// TIA Portal V20 program export: 2 tag tables, 2 data types, 3 data blocks, 5 code blocks (in call order from the OBs), 4 instance data blocks

VAR_GLOBAL   // PLC tag table "IO_Device_PCL_Centralilze_PLC_Functinal_Test_2"
   In_Test_Parameters AT %I100.0 : "IO_Device_Test_Parameters";
   Out_Functinal_Test AT %Q100.0 : "IO_Device_Functinal_Test";
END_VAR

VAR_GLOBAL   // PLC tag table "IO_PLC_Functinal_Test_2_PLC_Functinal_Test_4"
   In_Functional_Test AT %I300.0 : "IO_Device_Functinal_Test";
   Out_Test_Parameters AT %Q300.0 : "IO_Device_Test_Parameters";
END_VAR

TYPE "IO_Device_Functinal_Test"
   STRUCT
      Life_Trigger_PLC_Functional_Test_2 : Bool;
      Star_Test_PLC_Functional_Test_2 : Bool;
      Button_PLC_Functional_Test_2 : Bool;
      Electrical_Current_Test_Approved_PLC_Functional_Test_2 : Bool;
      Visual_Test_Approved_PLC_Functional_Test_2 : Bool;
      Electrical_Current_Read_PLC_Functional_Test_2 : UInt;
      Life_Trigger_PLC_Functional_Test_4 : Bool;
      Star_Test_PLC_Functional_Test_4 : Bool;
      Button_PLC_Functional_Test_4 : Bool;
      Electrical_Current_Test_Approved_PLC_Functional_Test_4 : Bool;
      Visual_Test_Approved_PLC_Functional_Test_4 : Bool;
      Electrical_Current_Read_PLC_Functional_Test_4 : UInt;
      Life_Trigger_PLC_Functional_Test_6 : Bool;
      Star_Test_PLC_Functional_Test_6 : Bool;
      Button_PLC_Functional_Test_6 : Bool;
      Electrical_Current_Test_Approved_PLC_Functional_Test_6 : Bool;
      Visual_Test_Approved_PLC_Functional_Test_6 : Bool;
      Electrical_Current_Read_PLC_Functional_Test_6 : UInt;
      Life_Trigger_PLC_Functional_Test_8 : Bool;
      Star_Test_PLC_Functional_Test_8 : Bool;
      Button_PLC_Functional_Test_8 : Bool;
      Electrical_Current_Test_Approved_PLC_Functional_Test_8 : Bool;
      Visual_Test_Approved_PLC_Functional_Test_8 : Bool;
      Electrical_Current_Read_PLC_Functional_Test_8 : UInt;
      Life_Trigger_PLC_Functional_Test_10 : Bool;
      Star_Test_PLC_Functional_Test_10 : Bool;
      Button_PLC_Functional_Test_10 : Bool;
      Electrical_Current_Test_Approved_PLC_Functional_Test_10 : Bool;
      Visual_Test_Approved_PLC_Functional_Test_10 : Bool;
      Electrical_Current_Read_PLC_Functional_Test_10 : UInt;
      Life_Trigger_PLC_Functional_Test_12 : Bool;
      Star_Test_PLC_Functional_Test_12 : Bool;
      Button_PLC_Functional_Test_12 : Bool;
      Electrical_Current_Test_Approved_PLC_Functional_Test_12 : Bool;
      Visual_Test_Approved_PLC_Functional_Test_12 : Bool;
      Electrical_Current_Read_PLC_Functional_Test_12 : UInt;
      Life_Trigger_PLC_Functional_Test_14 : Bool;
      Star_Test_PLC_Functional_Test_14 : Bool;
      Button_PLC_Functional_Test_14 : Bool;
      Electrical_Current_Test_Approved_PLC_Functional_Test_14 : Bool;
      Visual_Test_Approved_PLC_Functional_Test_14 : Bool;
      Electrical_Current_Read_PLC_Functional_Test_14 : UInt;
      Life_Trigger_PLC_Functional_Test_16 : Bool;
      Star_Test_PLC_Functional_Test_16 : Bool;
      Button_PLC_Functional_Test_16 : Bool;
      Electrical_Current_Test_Approved_PLC_Functional_Test_16 : Bool;
      Visual_Test_Approved_PLC_Functional_Test_16 : Bool;
      Electrical_Current_Read_PLC_Functional_Test_16 : UInt;
      Life_Trigger_PLC_Functional_Test_18 : Bool;
      Star_Test_PLC_Functional_Test_18 : Bool;
      Button_PLC_Functional_Test_18 : Bool;
      Electrical_Current_Test_Approved_PLC_Functional_Test_18 : Bool;
      Visual_Test_Approved_PLC_Functional_Test_18 : Bool;
      Electrical_Current_Read_PLC_Functional_Test_18 : UInt;
      Life_Trigger_PLC_Functional_Test_20 : Bool;
      Star_Test_PLC_Functional_Test_20 : Bool;
      Button_PLC_Functional_Test_20 : Bool;
      Electrical_Current_Test_Approved_PLC_Functional_Test_20 : Bool;
      Visual_Test_Approved_PLC_Functional_Test_20 : Bool;
      Electrical_Current_Read_PLC_Functional_Test_20 : UInt;
      Life_Trigger_PLC_Functional_Test_22 : Bool;
      Star_Test_PLC_Functional_Test_22 : Bool;
      Button_PLC_Functional_Test_22 : Bool;
      Electrical_Current_Test_Approved_PLC_Functional_Test_22 : Bool;
      Visual_Test_Approved_PLC_Functional_Test_22 : Bool;
      Electrical_Current_Read_PLC_Functional_Test_22 : UInt;
      Life_Trigger_PLC_Functional_Test_24 : Bool;
      Star_Test_PLC_Functional_Test_24 : Bool;
      Button_PLC_Functional_Test_24 : Bool;
      Electrical_Current_Test_Approved_PLC_Functional_Test_24 : Bool;
      Visual_Test_Approved_PLC_Functional_Test_24 : Bool;
      Electrical_Current_Read_PLC_Functional_Test_24 : UInt;
      Life_Trigger_PLC_Functional_Test_26 : Bool;
      Star_Test_PLC_Functional_Test_26 : Bool;
      Button_PLC_Functional_Test_26 : Bool;
      Electrical_Current_Test_Approved_PLC_Functional_Test_26 : Bool;
      Visual_Test_Approved_PLC_Functional_Test_26 : Bool;
      Electrical_Current_Read_PLC_Functional_Test_26 : UInt;
      Life_Trigger_PLC_Functional_Test_28 : Bool;
      Star_Test_PLC_Functional_Test_28 : Bool;
      Button_PLC_Functional_Test_28 : Bool;
      Electrical_Current_Test_Approved_PLC_Functional_Test_28 : Bool;
      Visual_Test_Approved_PLC_Functional_Test_28 : Bool;
      Electrical_Current_Read_PLC_Functional_Test_28 : UInt;
      Life_Trigger_PLC_Functional_Test_30 : Bool;
      Star_Test_PLC_Functional_Test_30 : Bool;
      Button_PLC_Functional_Test_30 : Bool;
      Electrical_Current_Test_Approved_PLC_Functional_Test_30 : Bool;
      Visual_Test_Approved_PLC_Functional_Test_30 : Bool;
      Electrical_Current_Read_PLC_Functional_Test_30 : UInt;
   END_STRUCT;
END_TYPE

TYPE "IO_Device_Test_Parameters"
   STRUCT
      Reset_PLC_Functional_Test_2 : Bool;
      Reset_PLC_Functional_Test_4 : Bool;
      Reset_PLC_Functional_Test_6 : Bool;
      Reset_PLC_Functional_Test_8 : Bool;
      Reset_PLC_Functional_Test_10 : Bool;
      Reset_PLC_Functional_Test_12 : Bool;
      Reset_PLC_Functional_Test_14 : Bool;
      Reset_PLC_Functional_Test_16 : Bool;
      Reset_PLC_Functional_Test_18 : Bool;
      Reset_PLC_Functional_Test_20 : Bool;
      Reset_PLC_Functional_Test_22 : Bool;
      Reset_PLC_Functional_Test_24 : Bool;
      Reset_PLC_Functional_Test_26 : Bool;
      Reset_PLC_Functional_Test_28 : Bool;
      Reset_PLC_Functional_Test_30 : Bool;
      Status : Bool;
      Voltage_Read : UInt;
      Min_Electrical_Current : UInt;
      Max_Electrical_Current : UInt;
      Time_End_Electrical_Current_Test : Time;
      Time_Start_Visual_Test : Time;
   END_STRUCT;
END_TYPE

DATA_BLOCK "DB_Analogic_Inputs"   // DB2
{ S7_Optimized_Access := 'TRUE' }
// stored: MemoryReserve 100
   VAR
      Electrical_Current_Read_Real : Real;
      Electrical_Voltage_Read_Real : Real;
      Electrical_Current_Read_UInt : UInt;
      Electrical_Voltage_Read_UInt : UInt;
   END_VAR
BEGIN
END_DATA_BLOCK

DATA_BLOCK "DB_Digital_Inputs"   // DB1
{ S7_Optimized_Access := 'TRUE' }
// stored: MemoryReserve 100
   VAR
      Button_Start_Approve : Bool;
      Digital_Input_1 : Bool;
      Digital_Input_2 : Bool;
      Digital_Input_3 : Bool;
      Digital_Input_4 : Bool;
      Digital_Input_5 : Bool;
   END_VAR
BEGIN
END_DATA_BLOCK

DATA_BLOCK "DB_Digital_Outputs"   // DB3
{ S7_Optimized_Access := 'TRUE' }
// stored: AutoNumber false, MemoryReserve 100
   VAR
      Blink_Button_Light : Bool;
      Turn_On_Button_Light : Bool;
      Light_Fail_Test : Bool;
      Light_Approve_Test : Bool;
      Digital_Output_3 : Bool;
   END_VAR
BEGIN
END_DATA_BLOCK

ORGANIZATION_BLOCK "Main"   // OB1, LAD, ProgramCycle
TITLE = "Main Program Sweep (Cycle)"
{ S7_Optimized_Access := 'TRUE' }
// stored: SetENOAutomatically false
   VAR_INPUT
      Initial_Call : Bool;   // Initial call of this OB
      Remanence : Bool;   // =True, if remanent data are available
   END_VAR
   VAR CONSTANT
      Test_Station : SInt := 2;
      Total_Number_Test_Stations : SInt := 25;
   END_VAR
BEGIN

REGION Network 1: Digital Inputs
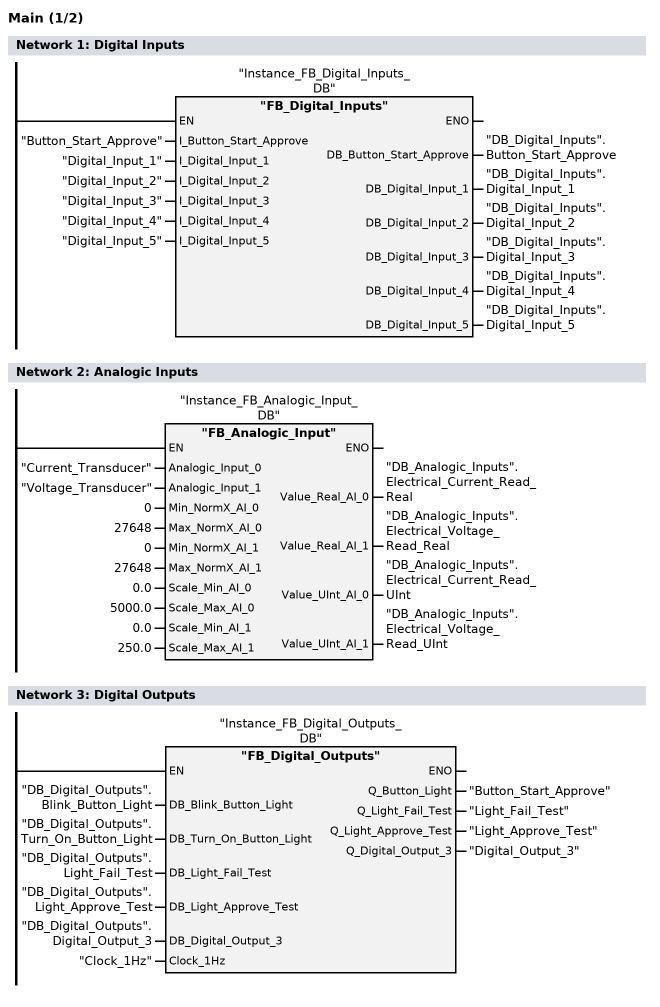
   RUNG wire#powerrail
      "Instance_FB_Digital_Inputs_DB"(I_Button_Start_Approve := "Button_Start_Approve", I_Digital_Input_1 := "Digital_Input_1", I_Digital_Input_2 := "Digital_Input_2", I_Digital_Input_3 := "Digital_Input_3", I_Digital_Input_4 := "Digital_Input_4", I_Digital_Input_5 := "Digital_Input_5", DB_Button_Start_Approve => "DB_Digital_Inputs".Button_Start_Approve, DB_Digital_Input_1 => "DB_Digital_Inputs".Digital_Input_1, DB_Digital_Input_2 => "DB_Digital_Inputs".Digital_Input_2, DB_Digital_Input_3 => "DB_Digital_Inputs".Digital_Input_3, DB_Digital_Input_4 => "DB_Digital_Inputs".Digital_Input_4, DB_Digital_Input_5 => "DB_Digital_Inputs".Digital_Input_5)
   END_RUNG
   // the same network as SCL:
   "Instance_FB_Digital_Inputs_DB"(I_Button_Start_Approve := "Button_Start_Approve",   // "FB_Digital_Inputs"
                           I_Digital_Input_1 := "Digital_Input_1",
                           I_Digital_Input_2 := "Digital_Input_2",
                           I_Digital_Input_3 := "Digital_Input_3",
                           I_Digital_Input_4 := "Digital_Input_4",
                           I_Digital_Input_5 := "Digital_Input_5",
                           DB_Button_Start_Approve => "DB_Digital_Inputs".Button_Start_Approve,
                           DB_Digital_Input_1 => "DB_Digital_Inputs".Digital_Input_1,
                           DB_Digital_Input_2 => "DB_Digital_Inputs".Digital_Input_2,
                           DB_Digital_Input_3 => "DB_Digital_Inputs".Digital_Input_3,
                           DB_Digital_Input_4 => "DB_Digital_Inputs".Digital_Input_4,
                           DB_Digital_Input_5 => "DB_Digital_Inputs".Digital_Input_5);
END_REGION

REGION Network 2: Analogic Inputs
   RUNG wire#powerrail
      "Instance_FB_Analogic_Input_DB"(Analogic_Input_0 := "Current_Transducer", Analogic_Input_1 := "Voltage_Transducer", Min_NormX_AI_0 := 0, Max_NormX_AI_0 := 27648, Min_NormX_AI_1 := 0, Max_NormX_AI_1 := 27648, Scale_Min_AI_0 := 0.0, Scale_Max_AI_0 := 5000.0, Scale_Min_AI_1 := 0.0, Scale_Max_AI_1 := 250.0, Value_Real_AI_0 => "DB_Analogic_Inputs".Electrical_Current_Read_Real, Value_Real_AI_1 => "DB_Analogic_Inputs".Electrical_Voltage_Read_Real, Value_UInt_AI_0 => "DB_Analogic_Inputs".Electrical_Current_Read_UInt, Value_UInt_AI_1 => "DB_Analogic_Inputs".Electrical_Voltage_Read_UInt)
   END_RUNG
   // the same network as SCL:
   "Instance_FB_Analogic_Input_DB"(Analogic_Input_0 := "Current_Transducer",   // "FB_Analogic_Input"
                           Analogic_Input_1 := "Voltage_Transducer",
                           Min_NormX_AI_0 := 0,
                           Max_NormX_AI_0 := 27648,
                           Min_NormX_AI_1 := 0,
                           Max_NormX_AI_1 := 27648,
                           Scale_Min_AI_0 := 0.0,
                           Scale_Max_AI_0 := 5000.0,
                           Scale_Min_AI_1 := 0.0,
                           Scale_Max_AI_1 := 250.0,
                           Value_Real_AI_0 => "DB_Analogic_Inputs".Electrical_Current_Read_Real,
                           Value_Real_AI_1 => "DB_Analogic_Inputs".Electrical_Voltage_Read_Real,
                           Value_UInt_AI_0 => "DB_Analogic_Inputs".Electrical_Current_Read_UInt,
                           Value_UInt_AI_1 => "DB_Analogic_Inputs".Electrical_Voltage_Read_UInt);
END_REGION

REGION Network 3: Digital Outputs
   RUNG wire#powerrail
      "Instance_FB_Digital_Outputs_DB"(DB_Blink_Button_Light := "DB_Digital_Outputs".Blink_Button_Light, DB_Turn_On_Button_Light := "DB_Digital_Outputs".Turn_On_Button_Light, DB_Light_Fail_Test := "DB_Digital_Outputs".Light_Fail_Test, DB_Light_Approve_Test := "DB_Digital_Outputs".Light_Approve_Test, DB_Digital_Output_3 := "DB_Digital_Outputs".Digital_Output_3, Clock_1Hz := "Clock_1Hz", Q_Button_Light => "Button_Start_Approve", Q_Light_Fail_Test => "Light_Fail_Test", Q_Light_Approve_Test => "Light_Approve_Test", Q_Digital_Output_3 => "Digital_Output_3")
   END_RUNG
   // the same network as SCL:
   "Instance_FB_Digital_Outputs_DB"(DB_Blink_Button_Light := "DB_Digital_Outputs".Blink_Button_Light,   // "FB_Digital_Outputs"
                           DB_Turn_On_Button_Light := "DB_Digital_Outputs".Turn_On_Button_Light,
                           DB_Light_Fail_Test := "DB_Digital_Outputs".Light_Fail_Test,
                           DB_Light_Approve_Test := "DB_Digital_Outputs".Light_Approve_Test,
                           DB_Digital_Output_3 := "DB_Digital_Outputs".Digital_Output_3,
                           Clock_1Hz := "Clock_1Hz",
                           Q_Button_Light => "Button_Start_Approve",
                           Q_Light_Fail_Test => "Light_Fail_Test",
                           Q_Light_Approve_Test => "Light_Approve_Test",
                           Q_Digital_Output_3 => "Digital_Output_3");
END_REGION

REGION Network 4: IO Device
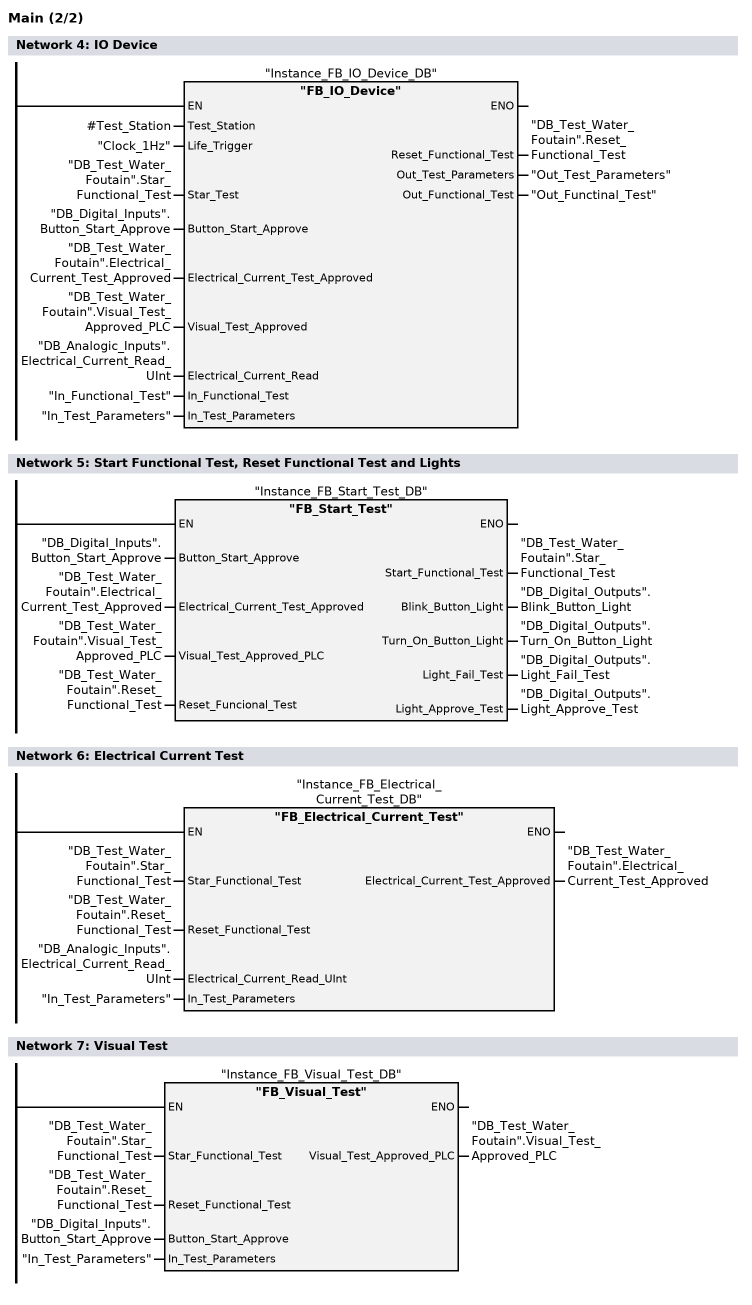
   RUNG wire#powerrail
      "Instance_FB_IO_Device_DB"(Test_Station := #Test_Station, Life_Trigger := "Clock_1Hz", Star_Test := "DB_Test_Water_Foutain".Star_Functional_Test, Button_Start_Approve := "DB_Digital_Inputs".Button_Start_Approve, Electrical_Current_Test_Approved := "DB_Test_Water_Foutain".Electrical_Current_Test_Approved, Visual_Test_Approved := "DB_Test_Water_Foutain".Visual_Test_Approved_PLC, Electrical_Current_Read := "DB_Analogic_Inputs".Electrical_Current_Read_UInt, In_Functional_Test := "In_Functional_Test", In_Test_Parameters := "In_Test_Parameters", Reset_Functional_Test => "DB_Test_Water_Foutain".Reset_Functional_Test, Out_Test_Parameters => "Out_Test_Parameters", Out_Functional_Test => "Out_Functinal_Test")
   END_RUNG
   // the same network as SCL:
   "Instance_FB_IO_Device_DB"(Test_Station := #Test_Station,   // "FB_IO_Device"
                           Life_Trigger := "Clock_1Hz",
                           Star_Test := "DB_Test_Water_Foutain".Star_Functional_Test,
                           Button_Start_Approve := "DB_Digital_Inputs".Button_Start_Approve,
                           Electrical_Current_Test_Approved := "DB_Test_Water_Foutain".Electrical_Current_Test_Approved,
                           Visual_Test_Approved := "DB_Test_Water_Foutain".Visual_Test_Approved_PLC,
                           Electrical_Current_Read := "DB_Analogic_Inputs".Electrical_Current_Read_UInt,
                           In_Functional_Test := "In_Functional_Test",
                           In_Test_Parameters := "In_Test_Parameters",
                           Reset_Functional_Test => "DB_Test_Water_Foutain".Reset_Functional_Test,
                           Out_Test_Parameters => "Out_Test_Parameters",
                           Out_Functional_Test => "Out_Functinal_Test");
END_REGION

REGION Network 5: Start Functional Test, Reset Functional Test and Lights
   RUNG wire#powerrail
      "Instance_FB_Start_Test_DB"(Button_Start_Approve := "DB_Digital_Inputs".Button_Start_Approve, Electrical_Current_Test_Approved := "DB_Test_Water_Foutain".Electrical_Current_Test_Approved, Visual_Test_Approved_PLC := "DB_Test_Water_Foutain".Visual_Test_Approved_PLC, Reset_Funcional_Test := "DB_Test_Water_Foutain".Reset_Functional_Test, Start_Functional_Test => "DB_Test_Water_Foutain".Star_Functional_Test, Blink_Button_Light => "DB_Digital_Outputs".Blink_Button_Light, Turn_On_Button_Light => "DB_Digital_Outputs".Turn_On_Button_Light, Light_Fail_Test => "DB_Digital_Outputs".Light_Fail_Test, Light_Approve_Test => "DB_Digital_Outputs".Light_Approve_Test)
   END_RUNG
   // the same network as SCL:
   "Instance_FB_Start_Test_DB"(Button_Start_Approve := "DB_Digital_Inputs".Button_Start_Approve,   // "FB_Start_Test"
                           Electrical_Current_Test_Approved := "DB_Test_Water_Foutain".Electrical_Current_Test_Approved,
                           Visual_Test_Approved_PLC := "DB_Test_Water_Foutain".Visual_Test_Approved_PLC,
                           Reset_Funcional_Test := "DB_Test_Water_Foutain".Reset_Functional_Test,
                           Start_Functional_Test => "DB_Test_Water_Foutain".Star_Functional_Test,
                           Blink_Button_Light => "DB_Digital_Outputs".Blink_Button_Light,
                           Turn_On_Button_Light => "DB_Digital_Outputs".Turn_On_Button_Light,
                           Light_Fail_Test => "DB_Digital_Outputs".Light_Fail_Test,
                           Light_Approve_Test => "DB_Digital_Outputs".Light_Approve_Test);
END_REGION

REGION Network 6: Electrical Current Test
   RUNG wire#powerrail
      "Instance_FB_Electrical_Current_Test_DB"(Star_Functional_Test := "DB_Test_Water_Foutain".Star_Functional_Test, Reset_Functional_Test := "DB_Test_Water_Foutain".Reset_Functional_Test, Electrical_Current_Read_UInt := "DB_Analogic_Inputs".Electrical_Current_Read_UInt, In_Test_Parameters := "In_Test_Parameters", Electrical_Current_Test_Approved => "DB_Test_Water_Foutain".Electrical_Current_Test_Approved)
   END_RUNG
   // the same network as SCL:
   "Instance_FB_Electrical_Current_Test_DB"(Star_Functional_Test := "DB_Test_Water_Foutain".Star_Functional_Test,   // "FB_Electrical_Current_Test"
                           Reset_Functional_Test := "DB_Test_Water_Foutain".Reset_Functional_Test,
                           Electrical_Current_Read_UInt := "DB_Analogic_Inputs".Electrical_Current_Read_UInt,
                           In_Test_Parameters := "In_Test_Parameters",
                           Electrical_Current_Test_Approved => "DB_Test_Water_Foutain".Electrical_Current_Test_Approved);
END_REGION

REGION Network 7: Visual Test
   RUNG wire#powerrail
      "Instance_FB_Visual_Test_DB"(Star_Functional_Test := "DB_Test_Water_Foutain".Star_Functional_Test, Reset_Functional_Test := "DB_Test_Water_Foutain".Reset_Functional_Test, Button_Start_Approve := "DB_Digital_Inputs".Button_Start_Approve, In_Test_Parameters := "In_Test_Parameters", Visual_Test_Approved_PLC => "DB_Test_Water_Foutain".Visual_Test_Approved_PLC)
   END_RUNG
   // the same network as SCL:
   "Instance_FB_Visual_Test_DB"(Star_Functional_Test := "DB_Test_Water_Foutain".Star_Functional_Test,   // "FB_Visual_Test"
                           Reset_Functional_Test := "DB_Test_Water_Foutain".Reset_Functional_Test,
                           Button_Start_Approve := "DB_Digital_Inputs".Button_Start_Approve,
                           In_Test_Parameters := "In_Test_Parameters",
                           Visual_Test_Approved_PLC => "DB_Test_Water_Foutain".Visual_Test_Approved_PLC);
END_REGION
END_ORGANIZATION_BLOCK

FUNCTION_BLOCK "FB_Digital_Inputs"   // FB1, LAD
{ S7_Optimized_Access := 'TRUE' }
// stored: MemoryReserve 100, SetENOAutomatically false
   VAR_INPUT
      I_Button_Start_Approve : Bool;
      I_Digital_Input_1 : Bool;
      I_Digital_Input_2 : Bool;
      I_Digital_Input_3 : Bool;
      I_Digital_Input_4 : Bool;
      I_Digital_Input_5 : Bool;
   END_VAR
   VAR_OUTPUT
      DB_Button_Start_Approve : Bool;
      DB_Digital_Input_1 : Bool;
      DB_Digital_Input_2 : Bool;
      DB_Digital_Input_3 : Bool;
      DB_Digital_Input_4 : Bool;
      DB_Digital_Input_5 : Bool;
   END_VAR
BEGIN

REGION Network 1
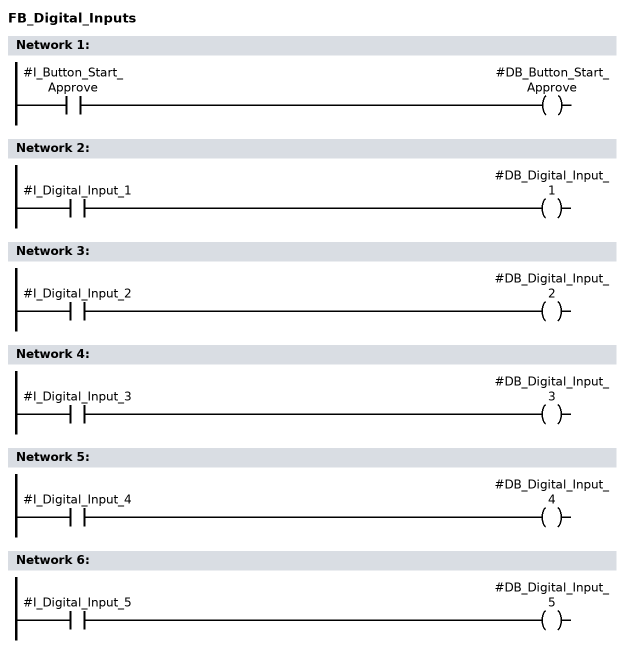
   RUNG wire#powerrail
      Contact( #I_Button_Start_Approve )
      Coil( #DB_Button_Start_Approve )
   END_RUNG
   // the same network as SCL:
   #DB_Button_Start_Approve := #I_Button_Start_Approve;
END_REGION

REGION Network 2
   RUNG wire#powerrail
      Contact( #I_Digital_Input_1 )
      Coil( #DB_Digital_Input_1 )
   END_RUNG
   // the same network as SCL:
   #DB_Digital_Input_1 := #I_Digital_Input_1;
END_REGION

REGION Network 3
   RUNG wire#powerrail
      Contact( #I_Digital_Input_2 )
      Coil( #DB_Digital_Input_2 )
   END_RUNG
   // the same network as SCL:
   #DB_Digital_Input_2 := #I_Digital_Input_2;
END_REGION

REGION Network 4
   RUNG wire#powerrail
      Contact( #I_Digital_Input_3 )
      Coil( #DB_Digital_Input_3 )
   END_RUNG
   // the same network as SCL:
   #DB_Digital_Input_3 := #I_Digital_Input_3;
END_REGION

REGION Network 5
   RUNG wire#powerrail
      Contact( #I_Digital_Input_4 )
      Coil( #DB_Digital_Input_4 )
   END_RUNG
   // the same network as SCL:
   #DB_Digital_Input_4 := #I_Digital_Input_4;
END_REGION

REGION Network 6
   RUNG wire#powerrail
      Contact( #I_Digital_Input_5 )
      Coil( #DB_Digital_Input_5 )
   END_RUNG
   // the same network as SCL:
   #DB_Digital_Input_5 := #I_Digital_Input_5;
END_REGION
END_FUNCTION_BLOCK

FUNCTION_BLOCK "FB_Digital_Outputs"   // FB3, LAD
{ S7_Optimized_Access := 'TRUE' }
// stored: AutoNumber false, MemoryReserve 100, SetENOAutomatically false
   VAR_INPUT
      DB_Blink_Button_Light : Bool;
      DB_Turn_On_Button_Light : Bool;
      DB_Light_Fail_Test : Bool;
      DB_Light_Approve_Test : Bool;
      DB_Digital_Output_3 : Bool;
      Clock_1Hz : Bool;
   END_VAR
   VAR_OUTPUT
      Q_Button_Light : Bool;
      Q_Light_Fail_Test : Bool;
      Q_Light_Approve_Test : Bool;
      Q_Digital_Output_3 : Bool;
   END_VAR
   VAR
      Timer_Delay_Fail_Test { S7_SetPoint := 'True'} : TON_TIME;
      Timer_Delay_Approve_Test { S7_SetPoint := 'True'} : TON_TIME;
   END_VAR
BEGIN

REGION Network 1
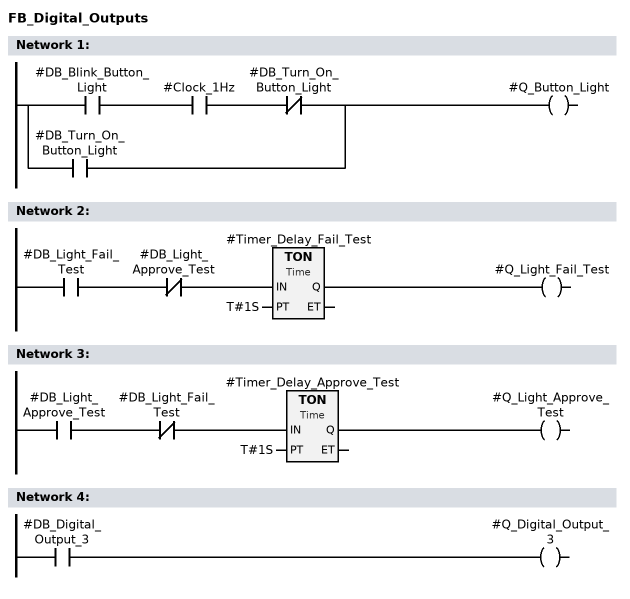
   RUNG wire#powerrail
      Contact( #DB_Blink_Button_Light )
      Contact( #Clock_1Hz )
      I_Contact( #DB_Turn_On_Button_Light )
      wire#w1
      Coil( #Q_Button_Light )
   END_RUNG
   RUNG wire#powerrail
      Contact( #DB_Turn_On_Button_Light )
   END_RUNG wire#w1
   // the same network as SCL:
   #Q_Button_Light := (#DB_Blink_Button_Light AND #Clock_1Hz AND NOT #DB_Turn_On_Button_Light) OR #DB_Turn_On_Button_Light;
END_REGION

REGION Network 2
   RUNG wire#powerrail
      Contact( #DB_Light_Fail_Test )
      I_Contact( #DB_Light_Approve_Test )
      { S7_Templates := "time_type := Time" } #Timer_Delay_Fail_Test.TON(pt := T#1S, et =>)
      Coil( #Q_Light_Fail_Test )
   END_RUNG
   // the same network as SCL:
   #Timer_Delay_Fail_Test(IN := #DB_Light_Fail_Test AND NOT #DB_Light_Approve_Test, PT := T#1S);   // TON
   #Q_Light_Fail_Test := #Timer_Delay_Fail_Test.Q;
END_REGION

REGION Network 3
   RUNG wire#powerrail
      Contact( #DB_Light_Approve_Test )
      I_Contact( #DB_Light_Fail_Test )
      { S7_Templates := "time_type := Time" } #Timer_Delay_Approve_Test.TON(pt := T#1S, et =>)
      Coil( #Q_Light_Approve_Test )
   END_RUNG
   // the same network as SCL:
   #Timer_Delay_Approve_Test(IN := #DB_Light_Approve_Test AND NOT #DB_Light_Fail_Test, PT := T#1S);   // TON
   #Q_Light_Approve_Test := #Timer_Delay_Approve_Test.Q;
END_REGION

REGION Network 4
   RUNG wire#powerrail
      Contact( #DB_Digital_Output_3 )
      Coil( #Q_Digital_Output_3 )
   END_RUNG
   // the same network as SCL:
   #Q_Digital_Output_3 := #DB_Digital_Output_3;
END_REGION
END_FUNCTION_BLOCK

FUNCTION_BLOCK "FB_IO_Device"   // FB4, LAD
{ S7_Optimized_Access := 'TRUE' }
// stored: MemoryReserve 100, SetENOAutomatically false
   VAR_INPUT
      Test_Station : SInt;
      Life_Trigger : Bool;
      Star_Test : Bool;
      Button_Start_Approve : Bool;
      Electrical_Current_Test_Approved : Bool;
      Visual_Test_Approved : Bool;
      Electrical_Current_Read : UInt;
      In_Functional_Test : "IO_Device_Functinal_Test";
      In_Test_Parameters : "IO_Device_Test_Parameters";
   END_VAR
   VAR_OUTPUT
      Reset_Functional_Test : Bool;
      Out_Test_Parameters : "IO_Device_Test_Parameters";
      Out_Functional_Test : "IO_Device_Functinal_Test";
   END_VAR
   VAR_TEMP   // added for the SCL form of the ladder/FBD networks
      _w1 : Bool;
   END_VAR
BEGIN

REGION Network 1: Test Parameters
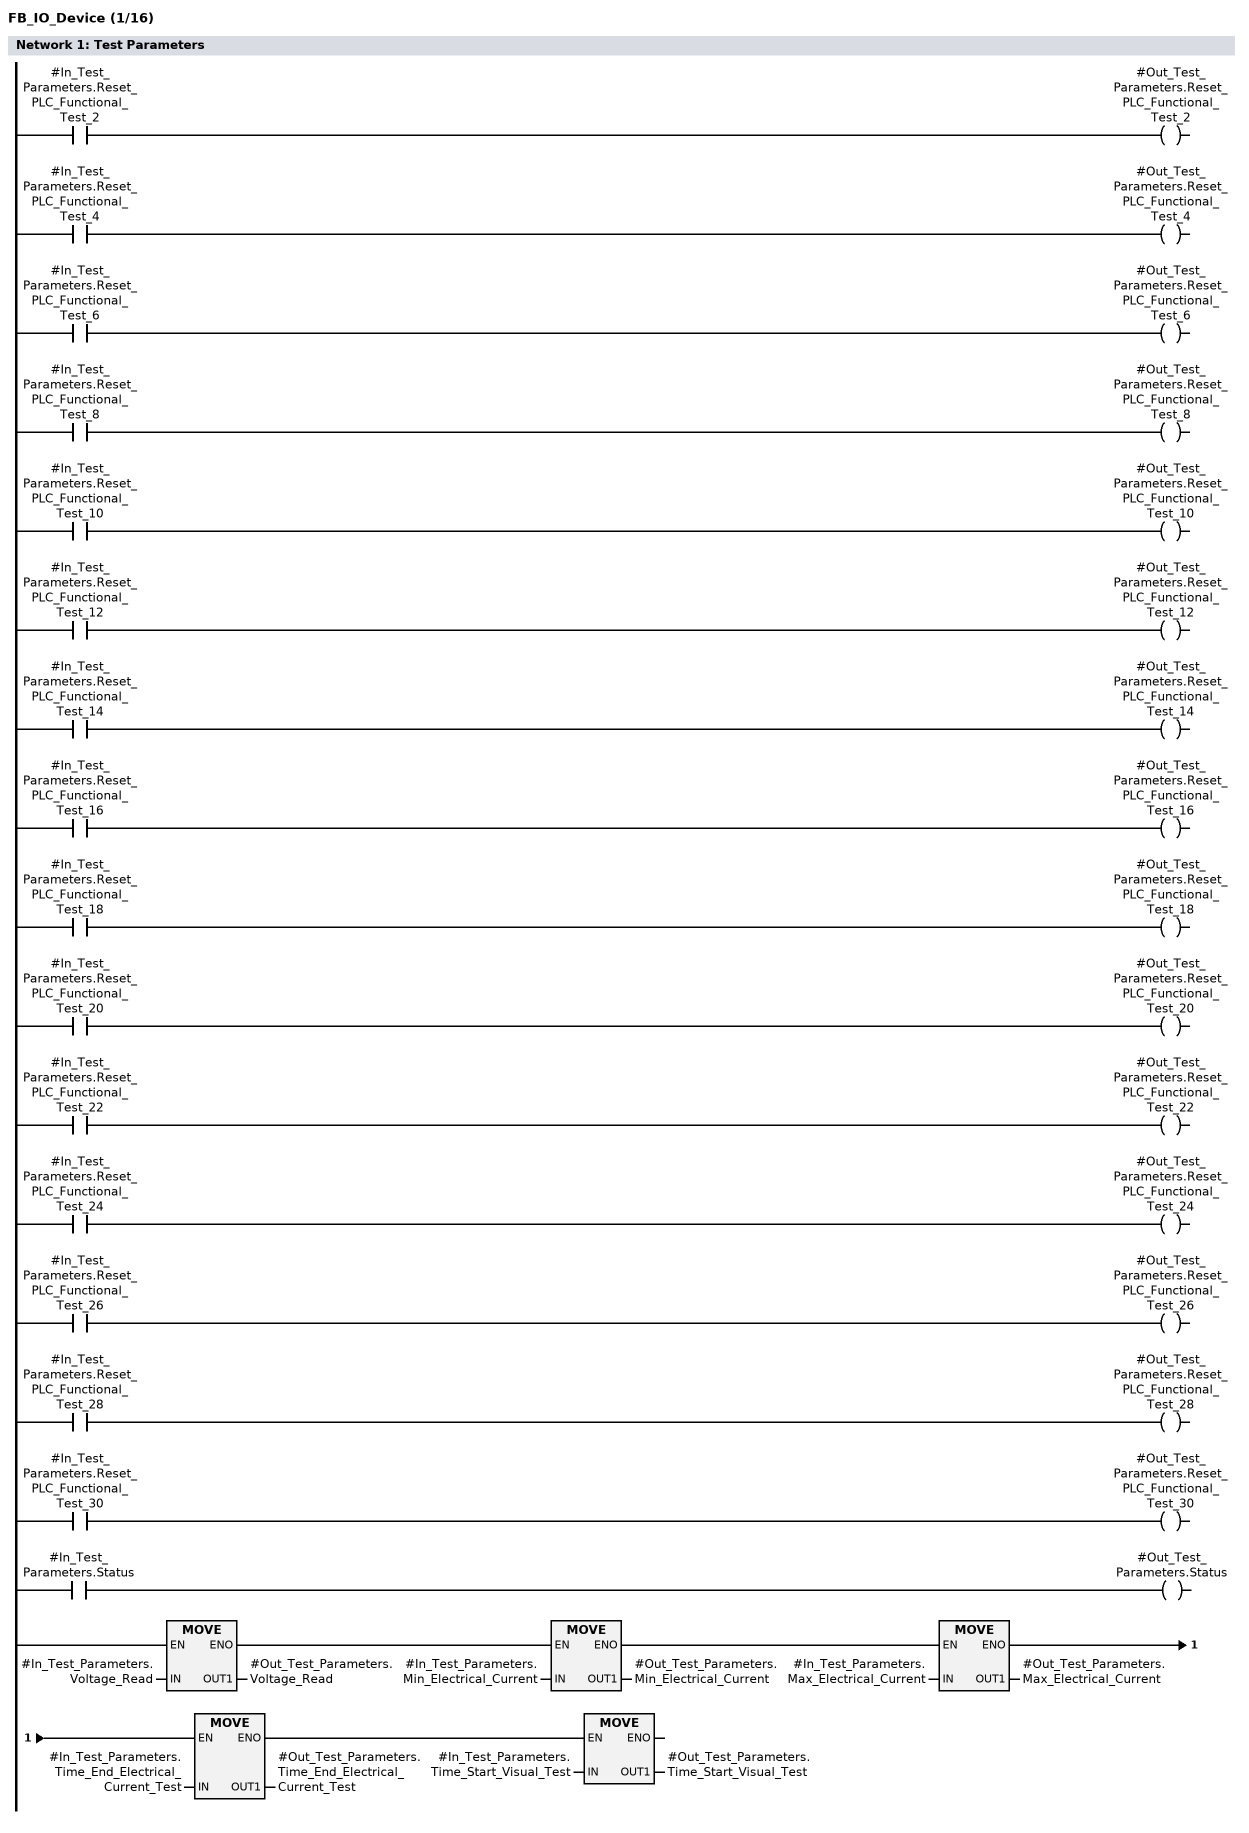
   RUNG wire#powerrail
      Contact( #In_Test_Parameters.Reset_PLC_Functional_Test_2 )
      Coil( #Out_Test_Parameters.Reset_PLC_Functional_Test_2 )
   END_RUNG
   RUNG wire#powerrail
      Contact( #In_Test_Parameters.Reset_PLC_Functional_Test_4 )
      Coil( #Out_Test_Parameters.Reset_PLC_Functional_Test_4 )
   END_RUNG
   RUNG wire#powerrail
      Contact( #In_Test_Parameters.Reset_PLC_Functional_Test_6 )
      Coil( #Out_Test_Parameters.Reset_PLC_Functional_Test_6 )
   END_RUNG
   RUNG wire#powerrail
      Contact( #In_Test_Parameters.Reset_PLC_Functional_Test_8 )
      Coil( #Out_Test_Parameters.Reset_PLC_Functional_Test_8 )
   END_RUNG
   RUNG wire#powerrail
      Contact( #In_Test_Parameters.Reset_PLC_Functional_Test_10 )
      Coil( #Out_Test_Parameters.Reset_PLC_Functional_Test_10 )
   END_RUNG
   RUNG wire#powerrail
      Contact( #In_Test_Parameters.Reset_PLC_Functional_Test_12 )
      Coil( #Out_Test_Parameters.Reset_PLC_Functional_Test_12 )
   END_RUNG
   RUNG wire#powerrail
      Contact( #In_Test_Parameters.Reset_PLC_Functional_Test_14 )
      Coil( #Out_Test_Parameters.Reset_PLC_Functional_Test_14 )
   END_RUNG
   RUNG wire#powerrail
      Contact( #In_Test_Parameters.Reset_PLC_Functional_Test_16 )
      Coil( #Out_Test_Parameters.Reset_PLC_Functional_Test_16 )
   END_RUNG
   RUNG wire#powerrail
      Contact( #In_Test_Parameters.Reset_PLC_Functional_Test_18 )
      Coil( #Out_Test_Parameters.Reset_PLC_Functional_Test_18 )
   END_RUNG
   RUNG wire#powerrail
      Contact( #In_Test_Parameters.Reset_PLC_Functional_Test_20 )
      Coil( #Out_Test_Parameters.Reset_PLC_Functional_Test_20 )
   END_RUNG
   RUNG wire#powerrail
      Contact( #In_Test_Parameters.Reset_PLC_Functional_Test_22 )
      Coil( #Out_Test_Parameters.Reset_PLC_Functional_Test_22 )
   END_RUNG
   RUNG wire#powerrail
      Contact( #In_Test_Parameters.Reset_PLC_Functional_Test_24 )
      Coil( #Out_Test_Parameters.Reset_PLC_Functional_Test_24 )
   END_RUNG
   RUNG wire#powerrail
      Contact( #In_Test_Parameters.Reset_PLC_Functional_Test_26 )
      Coil( #Out_Test_Parameters.Reset_PLC_Functional_Test_26 )
   END_RUNG
   RUNG wire#powerrail
      Contact( #In_Test_Parameters.Reset_PLC_Functional_Test_28 )
      Coil( #Out_Test_Parameters.Reset_PLC_Functional_Test_28 )
   END_RUNG
   RUNG wire#powerrail
      Contact( #In_Test_Parameters.Reset_PLC_Functional_Test_30 )
      Coil( #Out_Test_Parameters.Reset_PLC_Functional_Test_30 )
   END_RUNG
   RUNG wire#powerrail
      Contact( #In_Test_Parameters.Status )
      Coil( #Out_Test_Parameters.Status )
   END_RUNG
   RUNG wire#powerrail
      Move(in := #In_Test_Parameters.Voltage_Read, out1 => #Out_Test_Parameters.Voltage_Read)
      Move(in := #In_Test_Parameters.Min_Electrical_Current, out1 => #Out_Test_Parameters.Min_Electrical_Current)
      Move(in := #In_Test_Parameters.Max_Electrical_Current, out1 => #Out_Test_Parameters.Max_Electrical_Current)
      Move(in := #In_Test_Parameters.Time_End_Electrical_Current_Test, out1 => #Out_Test_Parameters.Time_End_Electrical_Current_Test)
      Move(in := #In_Test_Parameters.Time_Start_Visual_Test, out1 => #Out_Test_Parameters.Time_Start_Visual_Test)
   END_RUNG
   // the same network as SCL:
   #Out_Test_Parameters.Reset_PLC_Functional_Test_2 := #In_Test_Parameters.Reset_PLC_Functional_Test_2;
   #Out_Test_Parameters.Reset_PLC_Functional_Test_4 := #In_Test_Parameters.Reset_PLC_Functional_Test_4;
   #Out_Test_Parameters.Reset_PLC_Functional_Test_6 := #In_Test_Parameters.Reset_PLC_Functional_Test_6;
   #Out_Test_Parameters.Reset_PLC_Functional_Test_8 := #In_Test_Parameters.Reset_PLC_Functional_Test_8;
   #Out_Test_Parameters.Reset_PLC_Functional_Test_10 := #In_Test_Parameters.Reset_PLC_Functional_Test_10;
   #Out_Test_Parameters.Reset_PLC_Functional_Test_12 := #In_Test_Parameters.Reset_PLC_Functional_Test_12;
   #Out_Test_Parameters.Reset_PLC_Functional_Test_14 := #In_Test_Parameters.Reset_PLC_Functional_Test_14;
   #Out_Test_Parameters.Reset_PLC_Functional_Test_16 := #In_Test_Parameters.Reset_PLC_Functional_Test_16;
   #Out_Test_Parameters.Reset_PLC_Functional_Test_18 := #In_Test_Parameters.Reset_PLC_Functional_Test_18;
   #Out_Test_Parameters.Reset_PLC_Functional_Test_20 := #In_Test_Parameters.Reset_PLC_Functional_Test_20;
   #Out_Test_Parameters.Reset_PLC_Functional_Test_22 := #In_Test_Parameters.Reset_PLC_Functional_Test_22;
   #Out_Test_Parameters.Reset_PLC_Functional_Test_24 := #In_Test_Parameters.Reset_PLC_Functional_Test_24;
   #Out_Test_Parameters.Reset_PLC_Functional_Test_26 := #In_Test_Parameters.Reset_PLC_Functional_Test_26;
   #Out_Test_Parameters.Reset_PLC_Functional_Test_28 := #In_Test_Parameters.Reset_PLC_Functional_Test_28;
   #Out_Test_Parameters.Reset_PLC_Functional_Test_30 := #In_Test_Parameters.Reset_PLC_Functional_Test_30;
   #Out_Test_Parameters.Status := #In_Test_Parameters.Status;
   #Out_Test_Parameters.Voltage_Read := #In_Test_Parameters.Voltage_Read;
   #Out_Test_Parameters.Min_Electrical_Current := #In_Test_Parameters.Min_Electrical_Current;
   #Out_Test_Parameters.Max_Electrical_Current := #In_Test_Parameters.Max_Electrical_Current;
   #Out_Test_Parameters.Time_End_Electrical_Current_Test := #In_Test_Parameters.Time_End_Electrical_Current_Test;
   #Out_Test_Parameters.Time_Start_Visual_Test := #In_Test_Parameters.Time_Start_Visual_Test;
END_REGION

REGION Network 2: Functional Test Station 2
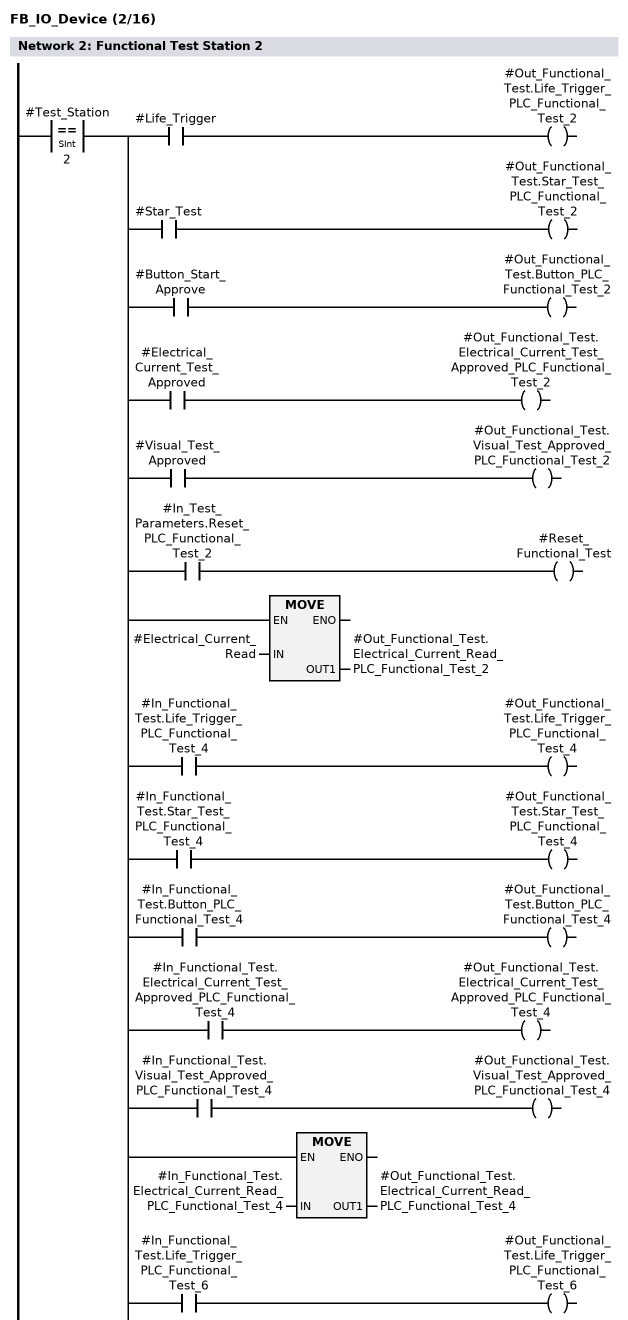
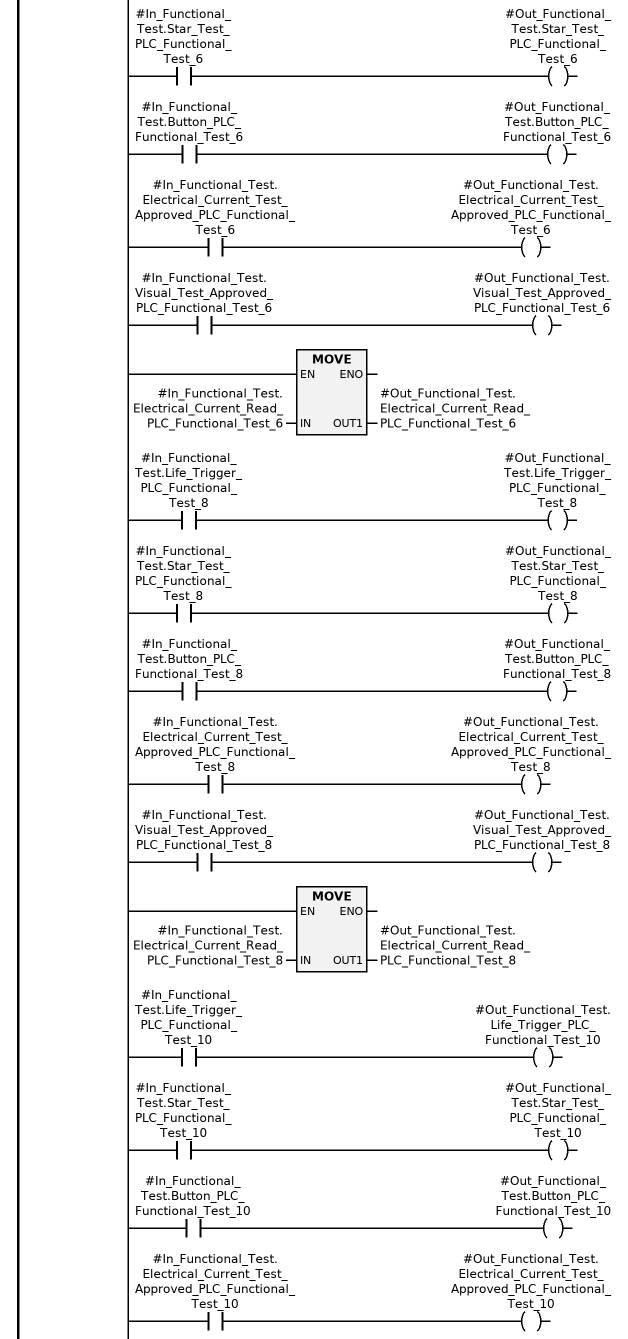
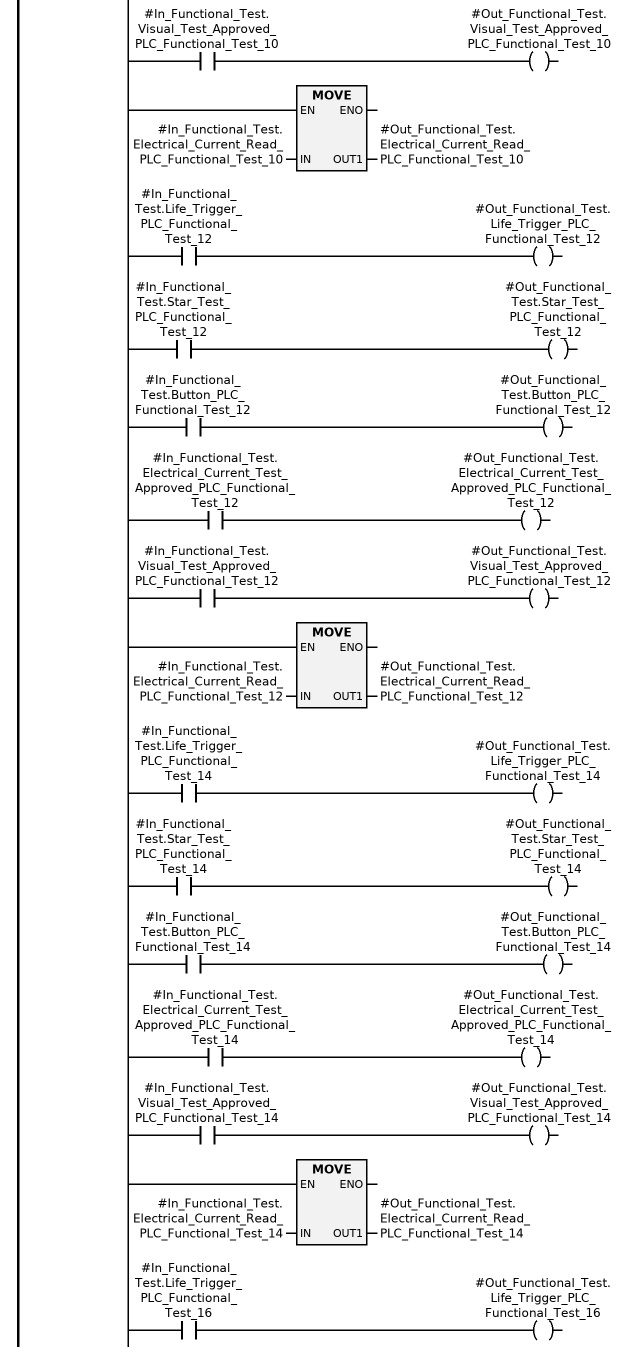
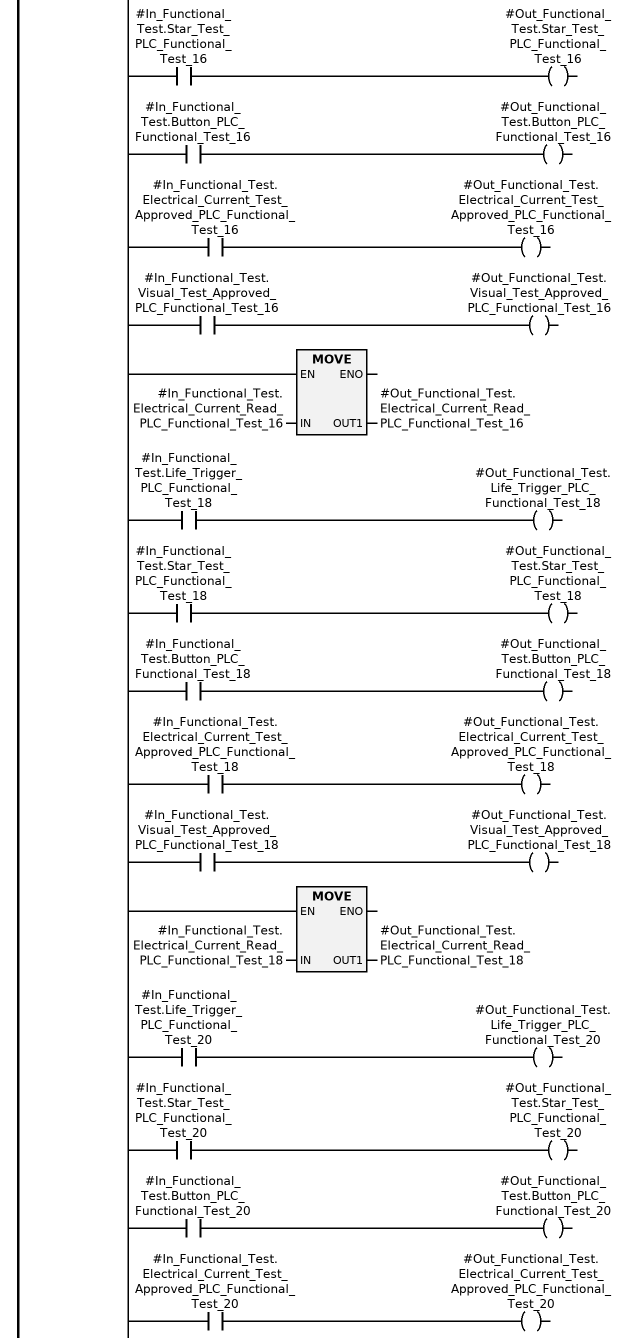
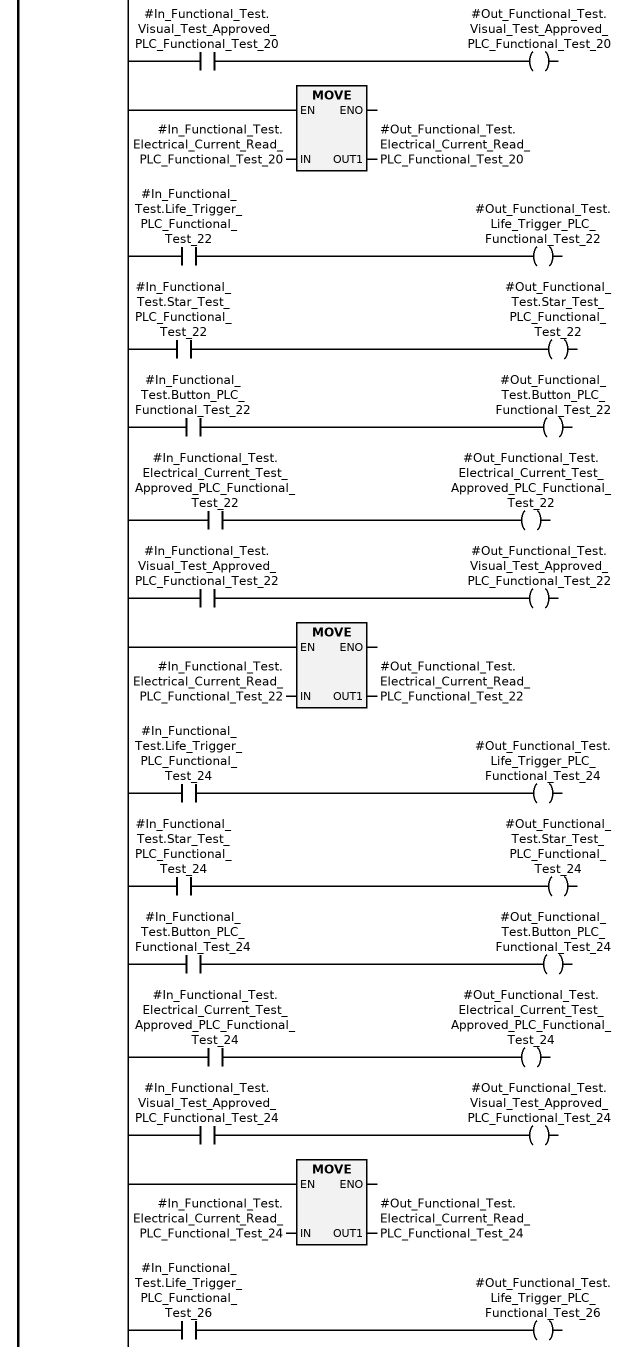
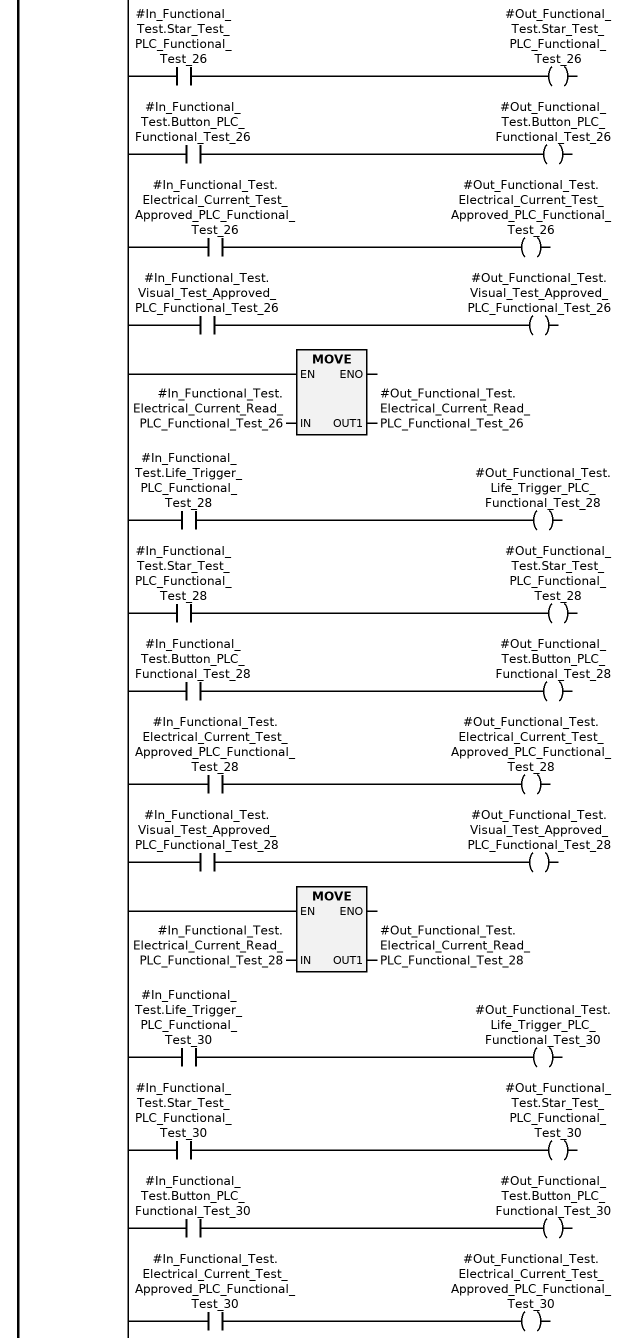
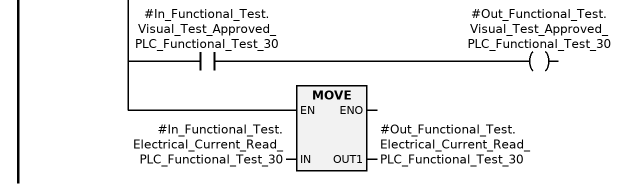
   RUNG wire#powerrail
      { S7_Templates := "SrcType := SInt" } EQ_Contact(in1 := #Test_Station, in2 := 2)
      wire#w1
      Contact( #Life_Trigger )
      Coil( #Out_Functional_Test.Life_Trigger_PLC_Functional_Test_2 )
   END_RUNG
   RUNG wire#w1
      Contact( #Star_Test )
      Coil( #Out_Functional_Test.Star_Test_PLC_Functional_Test_2 )
   END_RUNG
   RUNG wire#w1
      Contact( #Button_Start_Approve )
      Coil( #Out_Functional_Test.Button_PLC_Functional_Test_2 )
   END_RUNG
   RUNG wire#w1
      Contact( #Electrical_Current_Test_Approved )
      Coil( #Out_Functional_Test.Electrical_Current_Test_Approved_PLC_Functional_Test_2 )
   END_RUNG
   RUNG wire#w1
      Contact( #Visual_Test_Approved )
      Coil( #Out_Functional_Test.Visual_Test_Approved_PLC_Functional_Test_2 )
   END_RUNG
   RUNG wire#w1
      Contact( #In_Test_Parameters.Reset_PLC_Functional_Test_2 )
      Coil( #Reset_Functional_Test )
   END_RUNG
   RUNG wire#w1
      Move(in := #Electrical_Current_Read, out1 => #Out_Functional_Test.Electrical_Current_Read_PLC_Functional_Test_2)
   END_RUNG
   RUNG wire#w1
      Contact( #In_Functional_Test.Life_Trigger_PLC_Functional_Test_4 )
      Coil( #Out_Functional_Test.Life_Trigger_PLC_Functional_Test_4 )
   END_RUNG
   RUNG wire#w1
      Contact( #In_Functional_Test.Star_Test_PLC_Functional_Test_4 )
      Coil( #Out_Functional_Test.Star_Test_PLC_Functional_Test_4 )
   END_RUNG
   RUNG wire#w1
      Contact( #In_Functional_Test.Button_PLC_Functional_Test_4 )
      Coil( #Out_Functional_Test.Button_PLC_Functional_Test_4 )
   END_RUNG
   RUNG wire#w1
      Contact( #In_Functional_Test.Electrical_Current_Test_Approved_PLC_Functional_Test_4 )
      Coil( #Out_Functional_Test.Electrical_Current_Test_Approved_PLC_Functional_Test_4 )
   END_RUNG
   RUNG wire#w1
      Contact( #In_Functional_Test.Visual_Test_Approved_PLC_Functional_Test_4 )
      Coil( #Out_Functional_Test.Visual_Test_Approved_PLC_Functional_Test_4 )
   END_RUNG
   RUNG wire#w1
      Move(in := #In_Functional_Test.Electrical_Current_Read_PLC_Functional_Test_4, out1 => #Out_Functional_Test.Electrical_Current_Read_PLC_Functional_Test_4)
   END_RUNG
   RUNG wire#w1
      Contact( #In_Functional_Test.Life_Trigger_PLC_Functional_Test_6 )
      Coil( #Out_Functional_Test.Life_Trigger_PLC_Functional_Test_6 )
   END_RUNG
   RUNG wire#w1
      Contact( #In_Functional_Test.Star_Test_PLC_Functional_Test_6 )
      Coil( #Out_Functional_Test.Star_Test_PLC_Functional_Test_6 )
   END_RUNG
   RUNG wire#w1
      Contact( #In_Functional_Test.Button_PLC_Functional_Test_6 )
      Coil( #Out_Functional_Test.Button_PLC_Functional_Test_6 )
   END_RUNG
   RUNG wire#w1
      Contact( #In_Functional_Test.Electrical_Current_Test_Approved_PLC_Functional_Test_6 )
      Coil( #Out_Functional_Test.Electrical_Current_Test_Approved_PLC_Functional_Test_6 )
   END_RUNG
   RUNG wire#w1
      Contact( #In_Functional_Test.Visual_Test_Approved_PLC_Functional_Test_6 )
      Coil( #Out_Functional_Test.Visual_Test_Approved_PLC_Functional_Test_6 )
   END_RUNG
   RUNG wire#w1
      Move(in := #In_Functional_Test.Electrical_Current_Read_PLC_Functional_Test_6, out1 => #Out_Functional_Test.Electrical_Current_Read_PLC_Functional_Test_6)
   END_RUNG
   RUNG wire#w1
      Contact( #In_Functional_Test.Life_Trigger_PLC_Functional_Test_8 )
      Coil( #Out_Functional_Test.Life_Trigger_PLC_Functional_Test_8 )
   END_RUNG
   RUNG wire#w1
      Contact( #In_Functional_Test.Star_Test_PLC_Functional_Test_8 )
      Coil( #Out_Functional_Test.Star_Test_PLC_Functional_Test_8 )
   END_RUNG
   RUNG wire#w1
      Contact( #In_Functional_Test.Button_PLC_Functional_Test_8 )
      Coil( #Out_Functional_Test.Button_PLC_Functional_Test_8 )
   END_RUNG
   RUNG wire#w1
      Contact( #In_Functional_Test.Electrical_Current_Test_Approved_PLC_Functional_Test_8 )
      Coil( #Out_Functional_Test.Electrical_Current_Test_Approved_PLC_Functional_Test_8 )
   END_RUNG
   RUNG wire#w1
      Contact( #In_Functional_Test.Visual_Test_Approved_PLC_Functional_Test_8 )
      Coil( #Out_Functional_Test.Visual_Test_Approved_PLC_Functional_Test_8 )
   END_RUNG
   RUNG wire#w1
      Move(in := #In_Functional_Test.Electrical_Current_Read_PLC_Functional_Test_8, out1 => #Out_Functional_Test.Electrical_Current_Read_PLC_Functional_Test_8)
   END_RUNG
   RUNG wire#w1
      Contact( #In_Functional_Test.Life_Trigger_PLC_Functional_Test_10 )
      Coil( #Out_Functional_Test.Life_Trigger_PLC_Functional_Test_10 )
   END_RUNG
   RUNG wire#w1
      Contact( #In_Functional_Test.Star_Test_PLC_Functional_Test_10 )
      Coil( #Out_Functional_Test.Star_Test_PLC_Functional_Test_10 )
   END_RUNG
   RUNG wire#w1
      Contact( #In_Functional_Test.Button_PLC_Functional_Test_10 )
      Coil( #Out_Functional_Test.Button_PLC_Functional_Test_10 )
   END_RUNG
   RUNG wire#w1
      Contact( #In_Functional_Test.Electrical_Current_Test_Approved_PLC_Functional_Test_10 )
      Coil( #Out_Functional_Test.Electrical_Current_Test_Approved_PLC_Functional_Test_10 )
   END_RUNG
   RUNG wire#w1
      Contact( #In_Functional_Test.Visual_Test_Approved_PLC_Functional_Test_10 )
      Coil( #Out_Functional_Test.Visual_Test_Approved_PLC_Functional_Test_10 )
   END_RUNG
   RUNG wire#w1
      Move(in := #In_Functional_Test.Electrical_Current_Read_PLC_Functional_Test_10, out1 => #Out_Functional_Test.Electrical_Current_Read_PLC_Functional_Test_10)
   END_RUNG
   RUNG wire#w1
      Contact( #In_Functional_Test.Life_Trigger_PLC_Functional_Test_12 )
      Coil( #Out_Functional_Test.Life_Trigger_PLC_Functional_Test_12 )
   END_RUNG
   RUNG wire#w1
      Contact( #In_Functional_Test.Star_Test_PLC_Functional_Test_12 )
      Coil( #Out_Functional_Test.Star_Test_PLC_Functional_Test_12 )
   END_RUNG
   RUNG wire#w1
      Contact( #In_Functional_Test.Button_PLC_Functional_Test_12 )
      Coil( #Out_Functional_Test.Button_PLC_Functional_Test_12 )
   END_RUNG
   RUNG wire#w1
      Contact( #In_Functional_Test.Electrical_Current_Test_Approved_PLC_Functional_Test_12 )
      Coil( #Out_Functional_Test.Electrical_Current_Test_Approved_PLC_Functional_Test_12 )
   END_RUNG
   RUNG wire#w1
      Contact( #In_Functional_Test.Visual_Test_Approved_PLC_Functional_Test_12 )
      Coil( #Out_Functional_Test.Visual_Test_Approved_PLC_Functional_Test_12 )
   END_RUNG
   RUNG wire#w1
      Move(in := #In_Functional_Test.Electrical_Current_Read_PLC_Functional_Test_12, out1 => #Out_Functional_Test.Electrical_Current_Read_PLC_Functional_Test_12)
   END_RUNG
   RUNG wire#w1
      Contact( #In_Functional_Test.Life_Trigger_PLC_Functional_Test_14 )
      Coil( #Out_Functional_Test.Life_Trigger_PLC_Functional_Test_14 )
   END_RUNG
   RUNG wire#w1
      Contact( #In_Functional_Test.Star_Test_PLC_Functional_Test_14 )
      Coil( #Out_Functional_Test.Star_Test_PLC_Functional_Test_14 )
   END_RUNG
   RUNG wire#w1
      Contact( #In_Functional_Test.Button_PLC_Functional_Test_14 )
      Coil( #Out_Functional_Test.Button_PLC_Functional_Test_14 )
   END_RUNG
   RUNG wire#w1
      Contact( #In_Functional_Test.Electrical_Current_Test_Approved_PLC_Functional_Test_14 )
      Coil( #Out_Functional_Test.Electrical_Current_Test_Approved_PLC_Functional_Test_14 )
   END_RUNG
   RUNG wire#w1
      Contact( #In_Functional_Test.Visual_Test_Approved_PLC_Functional_Test_14 )
      Coil( #Out_Functional_Test.Visual_Test_Approved_PLC_Functional_Test_14 )
   END_RUNG
   RUNG wire#w1
      Move(in := #In_Functional_Test.Electrical_Current_Read_PLC_Functional_Test_14, out1 => #Out_Functional_Test.Electrical_Current_Read_PLC_Functional_Test_14)
   END_RUNG
   RUNG wire#w1
      Contact( #In_Functional_Test.Life_Trigger_PLC_Functional_Test_16 )
      Coil( #Out_Functional_Test.Life_Trigger_PLC_Functional_Test_16 )
   END_RUNG
   RUNG wire#w1
      Contact( #In_Functional_Test.Star_Test_PLC_Functional_Test_16 )
      Coil( #Out_Functional_Test.Star_Test_PLC_Functional_Test_16 )
   END_RUNG
   RUNG wire#w1
      Contact( #In_Functional_Test.Button_PLC_Functional_Test_16 )
      Coil( #Out_Functional_Test.Button_PLC_Functional_Test_16 )
   END_RUNG
   RUNG wire#w1
      Contact( #In_Functional_Test.Electrical_Current_Test_Approved_PLC_Functional_Test_16 )
      Coil( #Out_Functional_Test.Electrical_Current_Test_Approved_PLC_Functional_Test_16 )
   END_RUNG
   RUNG wire#w1
      Contact( #In_Functional_Test.Visual_Test_Approved_PLC_Functional_Test_16 )
      Coil( #Out_Functional_Test.Visual_Test_Approved_PLC_Functional_Test_16 )
   END_RUNG
   RUNG wire#w1
      Move(in := #In_Functional_Test.Electrical_Current_Read_PLC_Functional_Test_16, out1 => #Out_Functional_Test.Electrical_Current_Read_PLC_Functional_Test_16)
   END_RUNG
   RUNG wire#w1
      Contact( #In_Functional_Test.Life_Trigger_PLC_Functional_Test_18 )
      Coil( #Out_Functional_Test.Life_Trigger_PLC_Functional_Test_18 )
   END_RUNG
   RUNG wire#w1
      Contact( #In_Functional_Test.Star_Test_PLC_Functional_Test_18 )
      Coil( #Out_Functional_Test.Star_Test_PLC_Functional_Test_18 )
   END_RUNG
   RUNG wire#w1
      Contact( #In_Functional_Test.Button_PLC_Functional_Test_18 )
      Coil( #Out_Functional_Test.Button_PLC_Functional_Test_18 )
   END_RUNG
   RUNG wire#w1
      Contact( #In_Functional_Test.Electrical_Current_Test_Approved_PLC_Functional_Test_18 )
      Coil( #Out_Functional_Test.Electrical_Current_Test_Approved_PLC_Functional_Test_18 )
   END_RUNG
   RUNG wire#w1
      Contact( #In_Functional_Test.Visual_Test_Approved_PLC_Functional_Test_18 )
      Coil( #Out_Functional_Test.Visual_Test_Approved_PLC_Functional_Test_18 )
   END_RUNG
   RUNG wire#w1
      Move(in := #In_Functional_Test.Electrical_Current_Read_PLC_Functional_Test_18, out1 => #Out_Functional_Test.Electrical_Current_Read_PLC_Functional_Test_18)
   END_RUNG
   RUNG wire#w1
      Contact( #In_Functional_Test.Life_Trigger_PLC_Functional_Test_20 )
      Coil( #Out_Functional_Test.Life_Trigger_PLC_Functional_Test_20 )
   END_RUNG
   RUNG wire#w1
      Contact( #In_Functional_Test.Star_Test_PLC_Functional_Test_20 )
      Coil( #Out_Functional_Test.Star_Test_PLC_Functional_Test_20 )
   END_RUNG
   RUNG wire#w1
      Contact( #In_Functional_Test.Button_PLC_Functional_Test_20 )
      Coil( #Out_Functional_Test.Button_PLC_Functional_Test_20 )
   END_RUNG
   RUNG wire#w1
      Contact( #In_Functional_Test.Electrical_Current_Test_Approved_PLC_Functional_Test_20 )
      Coil( #Out_Functional_Test.Electrical_Current_Test_Approved_PLC_Functional_Test_20 )
   END_RUNG
   RUNG wire#w1
      Contact( #In_Functional_Test.Visual_Test_Approved_PLC_Functional_Test_20 )
      Coil( #Out_Functional_Test.Visual_Test_Approved_PLC_Functional_Test_20 )
   END_RUNG
   RUNG wire#w1
      Move(in := #In_Functional_Test.Electrical_Current_Read_PLC_Functional_Test_20, out1 => #Out_Functional_Test.Electrical_Current_Read_PLC_Functional_Test_20)
   END_RUNG
   RUNG wire#w1
      Contact( #In_Functional_Test.Life_Trigger_PLC_Functional_Test_22 )
      Coil( #Out_Functional_Test.Life_Trigger_PLC_Functional_Test_22 )
   END_RUNG
   RUNG wire#w1
      Contact( #In_Functional_Test.Star_Test_PLC_Functional_Test_22 )
      Coil( #Out_Functional_Test.Star_Test_PLC_Functional_Test_22 )
   END_RUNG
   RUNG wire#w1
      Contact( #In_Functional_Test.Button_PLC_Functional_Test_22 )
      Coil( #Out_Functional_Test.Button_PLC_Functional_Test_22 )
   END_RUNG
   RUNG wire#w1
      Contact( #In_Functional_Test.Electrical_Current_Test_Approved_PLC_Functional_Test_22 )
      Coil( #Out_Functional_Test.Electrical_Current_Test_Approved_PLC_Functional_Test_22 )
   END_RUNG
   RUNG wire#w1
      Contact( #In_Functional_Test.Visual_Test_Approved_PLC_Functional_Test_22 )
      Coil( #Out_Functional_Test.Visual_Test_Approved_PLC_Functional_Test_22 )
   END_RUNG
   RUNG wire#w1
      Move(in := #In_Functional_Test.Electrical_Current_Read_PLC_Functional_Test_22, out1 => #Out_Functional_Test.Electrical_Current_Read_PLC_Functional_Test_22)
   END_RUNG
   RUNG wire#w1
      Contact( #In_Functional_Test.Life_Trigger_PLC_Functional_Test_24 )
      Coil( #Out_Functional_Test.Life_Trigger_PLC_Functional_Test_24 )
   END_RUNG
   RUNG wire#w1
      Contact( #In_Functional_Test.Star_Test_PLC_Functional_Test_24 )
      Coil( #Out_Functional_Test.Star_Test_PLC_Functional_Test_24 )
   END_RUNG
   RUNG wire#w1
      Contact( #In_Functional_Test.Button_PLC_Functional_Test_24 )
      Coil( #Out_Functional_Test.Button_PLC_Functional_Test_24 )
   END_RUNG
   RUNG wire#w1
      Contact( #In_Functional_Test.Electrical_Current_Test_Approved_PLC_Functional_Test_24 )
      Coil( #Out_Functional_Test.Electrical_Current_Test_Approved_PLC_Functional_Test_24 )
   END_RUNG
   RUNG wire#w1
      Contact( #In_Functional_Test.Visual_Test_Approved_PLC_Functional_Test_24 )
      Coil( #Out_Functional_Test.Visual_Test_Approved_PLC_Functional_Test_24 )
   END_RUNG
   RUNG wire#w1
      Move(in := #In_Functional_Test.Electrical_Current_Read_PLC_Functional_Test_24, out1 => #Out_Functional_Test.Electrical_Current_Read_PLC_Functional_Test_24)
   END_RUNG
   RUNG wire#w1
      Contact( #In_Functional_Test.Life_Trigger_PLC_Functional_Test_26 )
      Coil( #Out_Functional_Test.Life_Trigger_PLC_Functional_Test_26 )
   END_RUNG
   RUNG wire#w1
      Contact( #In_Functional_Test.Star_Test_PLC_Functional_Test_26 )
      Coil( #Out_Functional_Test.Star_Test_PLC_Functional_Test_26 )
   END_RUNG
   RUNG wire#w1
      Contact( #In_Functional_Test.Button_PLC_Functional_Test_26 )
      Coil( #Out_Functional_Test.Button_PLC_Functional_Test_26 )
   END_RUNG
   RUNG wire#w1
      Contact( #In_Functional_Test.Electrical_Current_Test_Approved_PLC_Functional_Test_26 )
      Coil( #Out_Functional_Test.Electrical_Current_Test_Approved_PLC_Functional_Test_26 )
   END_RUNG
   RUNG wire#w1
      Contact( #In_Functional_Test.Visual_Test_Approved_PLC_Functional_Test_26 )
      Coil( #Out_Functional_Test.Visual_Test_Approved_PLC_Functional_Test_26 )
   END_RUNG
   RUNG wire#w1
      Move(in := #In_Functional_Test.Electrical_Current_Read_PLC_Functional_Test_26, out1 => #Out_Functional_Test.Electrical_Current_Read_PLC_Functional_Test_26)
   END_RUNG
   RUNG wire#w1
      Contact( #In_Functional_Test.Life_Trigger_PLC_Functional_Test_28 )
      Coil( #Out_Functional_Test.Life_Trigger_PLC_Functional_Test_28 )
   END_RUNG
   RUNG wire#w1
      Contact( #In_Functional_Test.Star_Test_PLC_Functional_Test_28 )
      Coil( #Out_Functional_Test.Star_Test_PLC_Functional_Test_28 )
   END_RUNG
   RUNG wire#w1
      Contact( #In_Functional_Test.Button_PLC_Functional_Test_28 )
      Coil( #Out_Functional_Test.Button_PLC_Functional_Test_28 )
   END_RUNG
   RUNG wire#w1
      Contact( #In_Functional_Test.Electrical_Current_Test_Approved_PLC_Functional_Test_28 )
      Coil( #Out_Functional_Test.Electrical_Current_Test_Approved_PLC_Functional_Test_28 )
   END_RUNG
   RUNG wire#w1
      Contact( #In_Functional_Test.Visual_Test_Approved_PLC_Functional_Test_28 )
      Coil( #Out_Functional_Test.Visual_Test_Approved_PLC_Functional_Test_28 )
   END_RUNG
   RUNG wire#w1
      Move(in := #In_Functional_Test.Electrical_Current_Read_PLC_Functional_Test_28, out1 => #Out_Functional_Test.Electrical_Current_Read_PLC_Functional_Test_28)
   END_RUNG
   RUNG wire#w1
      Contact( #In_Functional_Test.Life_Trigger_PLC_Functional_Test_30 )
      Coil( #Out_Functional_Test.Life_Trigger_PLC_Functional_Test_30 )
   END_RUNG
   RUNG wire#w1
      Contact( #In_Functional_Test.Star_Test_PLC_Functional_Test_30 )
      Coil( #Out_Functional_Test.Star_Test_PLC_Functional_Test_30 )
   END_RUNG
   RUNG wire#w1
      Contact( #In_Functional_Test.Button_PLC_Functional_Test_30 )
      Coil( #Out_Functional_Test.Button_PLC_Functional_Test_30 )
   END_RUNG
   RUNG wire#w1
      Contact( #In_Functional_Test.Electrical_Current_Test_Approved_PLC_Functional_Test_30 )
      Coil( #Out_Functional_Test.Electrical_Current_Test_Approved_PLC_Functional_Test_30 )
   END_RUNG
   RUNG wire#w1
      Contact( #In_Functional_Test.Visual_Test_Approved_PLC_Functional_Test_30 )
      Coil( #Out_Functional_Test.Visual_Test_Approved_PLC_Functional_Test_30 )
   END_RUNG
   RUNG wire#w1
      Move(in := #In_Functional_Test.Electrical_Current_Read_PLC_Functional_Test_30, out1 => #Out_Functional_Test.Electrical_Current_Read_PLC_Functional_Test_30)
   END_RUNG
   // the same network as SCL:
   #_w1 := #Test_Station = 2;
   #Out_Functional_Test.Life_Trigger_PLC_Functional_Test_2 := #_w1 AND #Life_Trigger;
   #Out_Functional_Test.Star_Test_PLC_Functional_Test_2 := #_w1 AND #Star_Test;
   #Out_Functional_Test.Button_PLC_Functional_Test_2 := #_w1 AND #Button_Start_Approve;
   #Out_Functional_Test.Electrical_Current_Test_Approved_PLC_Functional_Test_2 := #_w1 AND #Electrical_Current_Test_Approved;
   #Out_Functional_Test.Visual_Test_Approved_PLC_Functional_Test_2 := #_w1 AND #Visual_Test_Approved;
   #Reset_Functional_Test := #_w1 AND #In_Test_Parameters.Reset_PLC_Functional_Test_2;
   IF #_w1 THEN
       #Out_Functional_Test.Electrical_Current_Read_PLC_Functional_Test_2 := #Electrical_Current_Read;
   END_IF;
   #Out_Functional_Test.Life_Trigger_PLC_Functional_Test_4 := #_w1 AND #In_Functional_Test.Life_Trigger_PLC_Functional_Test_4;
   #Out_Functional_Test.Star_Test_PLC_Functional_Test_4 := #_w1 AND #In_Functional_Test.Star_Test_PLC_Functional_Test_4;
   #Out_Functional_Test.Button_PLC_Functional_Test_4 := #_w1 AND #In_Functional_Test.Button_PLC_Functional_Test_4;
   #Out_Functional_Test.Electrical_Current_Test_Approved_PLC_Functional_Test_4 := #_w1 AND #In_Functional_Test.Electrical_Current_Test_Approved_PLC_Functional_Test_4;
   #Out_Functional_Test.Visual_Test_Approved_PLC_Functional_Test_4 := #_w1 AND #In_Functional_Test.Visual_Test_Approved_PLC_Functional_Test_4;
   IF #_w1 THEN
       #Out_Functional_Test.Electrical_Current_Read_PLC_Functional_Test_4 := #In_Functional_Test.Electrical_Current_Read_PLC_Functional_Test_4;
   END_IF;
   #Out_Functional_Test.Life_Trigger_PLC_Functional_Test_6 := #_w1 AND #In_Functional_Test.Life_Trigger_PLC_Functional_Test_6;
   #Out_Functional_Test.Star_Test_PLC_Functional_Test_6 := #_w1 AND #In_Functional_Test.Star_Test_PLC_Functional_Test_6;
   #Out_Functional_Test.Button_PLC_Functional_Test_6 := #_w1 AND #In_Functional_Test.Button_PLC_Functional_Test_6;
   #Out_Functional_Test.Electrical_Current_Test_Approved_PLC_Functional_Test_6 := #_w1 AND #In_Functional_Test.Electrical_Current_Test_Approved_PLC_Functional_Test_6;
   #Out_Functional_Test.Visual_Test_Approved_PLC_Functional_Test_6 := #_w1 AND #In_Functional_Test.Visual_Test_Approved_PLC_Functional_Test_6;
   IF #_w1 THEN
       #Out_Functional_Test.Electrical_Current_Read_PLC_Functional_Test_6 := #In_Functional_Test.Electrical_Current_Read_PLC_Functional_Test_6;
   END_IF;
   #Out_Functional_Test.Life_Trigger_PLC_Functional_Test_8 := #_w1 AND #In_Functional_Test.Life_Trigger_PLC_Functional_Test_8;
   #Out_Functional_Test.Star_Test_PLC_Functional_Test_8 := #_w1 AND #In_Functional_Test.Star_Test_PLC_Functional_Test_8;
   #Out_Functional_Test.Button_PLC_Functional_Test_8 := #_w1 AND #In_Functional_Test.Button_PLC_Functional_Test_8;
   #Out_Functional_Test.Electrical_Current_Test_Approved_PLC_Functional_Test_8 := #_w1 AND #In_Functional_Test.Electrical_Current_Test_Approved_PLC_Functional_Test_8;
   #Out_Functional_Test.Visual_Test_Approved_PLC_Functional_Test_8 := #_w1 AND #In_Functional_Test.Visual_Test_Approved_PLC_Functional_Test_8;
   IF #_w1 THEN
       #Out_Functional_Test.Electrical_Current_Read_PLC_Functional_Test_8 := #In_Functional_Test.Electrical_Current_Read_PLC_Functional_Test_8;
   END_IF;
   #Out_Functional_Test.Life_Trigger_PLC_Functional_Test_10 := #_w1 AND #In_Functional_Test.Life_Trigger_PLC_Functional_Test_10;
   #Out_Functional_Test.Star_Test_PLC_Functional_Test_10 := #_w1 AND #In_Functional_Test.Star_Test_PLC_Functional_Test_10;
   #Out_Functional_Test.Button_PLC_Functional_Test_10 := #_w1 AND #In_Functional_Test.Button_PLC_Functional_Test_10;
   #Out_Functional_Test.Electrical_Current_Test_Approved_PLC_Functional_Test_10 := #_w1 AND #In_Functional_Test.Electrical_Current_Test_Approved_PLC_Functional_Test_10;
   #Out_Functional_Test.Visual_Test_Approved_PLC_Functional_Test_10 := #_w1 AND #In_Functional_Test.Visual_Test_Approved_PLC_Functional_Test_10;
   IF #_w1 THEN
       #Out_Functional_Test.Electrical_Current_Read_PLC_Functional_Test_10 := #In_Functional_Test.Electrical_Current_Read_PLC_Functional_Test_10;
   END_IF;
   #Out_Functional_Test.Life_Trigger_PLC_Functional_Test_12 := #_w1 AND #In_Functional_Test.Life_Trigger_PLC_Functional_Test_12;
   #Out_Functional_Test.Star_Test_PLC_Functional_Test_12 := #_w1 AND #In_Functional_Test.Star_Test_PLC_Functional_Test_12;
   #Out_Functional_Test.Button_PLC_Functional_Test_12 := #_w1 AND #In_Functional_Test.Button_PLC_Functional_Test_12;
   #Out_Functional_Test.Electrical_Current_Test_Approved_PLC_Functional_Test_12 := #_w1 AND #In_Functional_Test.Electrical_Current_Test_Approved_PLC_Functional_Test_12;
   #Out_Functional_Test.Visual_Test_Approved_PLC_Functional_Test_12 := #_w1 AND #In_Functional_Test.Visual_Test_Approved_PLC_Functional_Test_12;
   IF #_w1 THEN
       #Out_Functional_Test.Electrical_Current_Read_PLC_Functional_Test_12 := #In_Functional_Test.Electrical_Current_Read_PLC_Functional_Test_12;
   END_IF;
   #Out_Functional_Test.Life_Trigger_PLC_Functional_Test_14 := #_w1 AND #In_Functional_Test.Life_Trigger_PLC_Functional_Test_14;
   #Out_Functional_Test.Star_Test_PLC_Functional_Test_14 := #_w1 AND #In_Functional_Test.Star_Test_PLC_Functional_Test_14;
   #Out_Functional_Test.Button_PLC_Functional_Test_14 := #_w1 AND #In_Functional_Test.Button_PLC_Functional_Test_14;
   #Out_Functional_Test.Electrical_Current_Test_Approved_PLC_Functional_Test_14 := #_w1 AND #In_Functional_Test.Electrical_Current_Test_Approved_PLC_Functional_Test_14;
   #Out_Functional_Test.Visual_Test_Approved_PLC_Functional_Test_14 := #_w1 AND #In_Functional_Test.Visual_Test_Approved_PLC_Functional_Test_14;
   IF #_w1 THEN
       #Out_Functional_Test.Electrical_Current_Read_PLC_Functional_Test_14 := #In_Functional_Test.Electrical_Current_Read_PLC_Functional_Test_14;
   END_IF;
   #Out_Functional_Test.Life_Trigger_PLC_Functional_Test_16 := #_w1 AND #In_Functional_Test.Life_Trigger_PLC_Functional_Test_16;
   #Out_Functional_Test.Star_Test_PLC_Functional_Test_16 := #_w1 AND #In_Functional_Test.Star_Test_PLC_Functional_Test_16;
   #Out_Functional_Test.Button_PLC_Functional_Test_16 := #_w1 AND #In_Functional_Test.Button_PLC_Functional_Test_16;
   #Out_Functional_Test.Electrical_Current_Test_Approved_PLC_Functional_Test_16 := #_w1 AND #In_Functional_Test.Electrical_Current_Test_Approved_PLC_Functional_Test_16;
   #Out_Functional_Test.Visual_Test_Approved_PLC_Functional_Test_16 := #_w1 AND #In_Functional_Test.Visual_Test_Approved_PLC_Functional_Test_16;
   IF #_w1 THEN
       #Out_Functional_Test.Electrical_Current_Read_PLC_Functional_Test_16 := #In_Functional_Test.Electrical_Current_Read_PLC_Functional_Test_16;
   END_IF;
   #Out_Functional_Test.Life_Trigger_PLC_Functional_Test_18 := #_w1 AND #In_Functional_Test.Life_Trigger_PLC_Functional_Test_18;
   #Out_Functional_Test.Star_Test_PLC_Functional_Test_18 := #_w1 AND #In_Functional_Test.Star_Test_PLC_Functional_Test_18;
   #Out_Functional_Test.Button_PLC_Functional_Test_18 := #_w1 AND #In_Functional_Test.Button_PLC_Functional_Test_18;
   #Out_Functional_Test.Electrical_Current_Test_Approved_PLC_Functional_Test_18 := #_w1 AND #In_Functional_Test.Electrical_Current_Test_Approved_PLC_Functional_Test_18;
   #Out_Functional_Test.Visual_Test_Approved_PLC_Functional_Test_18 := #_w1 AND #In_Functional_Test.Visual_Test_Approved_PLC_Functional_Test_18;
   IF #_w1 THEN
       #Out_Functional_Test.Electrical_Current_Read_PLC_Functional_Test_18 := #In_Functional_Test.Electrical_Current_Read_PLC_Functional_Test_18;
   END_IF;
   #Out_Functional_Test.Life_Trigger_PLC_Functional_Test_20 := #_w1 AND #In_Functional_Test.Life_Trigger_PLC_Functional_Test_20;
   #Out_Functional_Test.Star_Test_PLC_Functional_Test_20 := #_w1 AND #In_Functional_Test.Star_Test_PLC_Functional_Test_20;
   #Out_Functional_Test.Button_PLC_Functional_Test_20 := #_w1 AND #In_Functional_Test.Button_PLC_Functional_Test_20;
   #Out_Functional_Test.Electrical_Current_Test_Approved_PLC_Functional_Test_20 := #_w1 AND #In_Functional_Test.Electrical_Current_Test_Approved_PLC_Functional_Test_20;
   #Out_Functional_Test.Visual_Test_Approved_PLC_Functional_Test_20 := #_w1 AND #In_Functional_Test.Visual_Test_Approved_PLC_Functional_Test_20;
   IF #_w1 THEN
       #Out_Functional_Test.Electrical_Current_Read_PLC_Functional_Test_20 := #In_Functional_Test.Electrical_Current_Read_PLC_Functional_Test_20;
   END_IF;
   #Out_Functional_Test.Life_Trigger_PLC_Functional_Test_22 := #_w1 AND #In_Functional_Test.Life_Trigger_PLC_Functional_Test_22;
   #Out_Functional_Test.Star_Test_PLC_Functional_Test_22 := #_w1 AND #In_Functional_Test.Star_Test_PLC_Functional_Test_22;
   #Out_Functional_Test.Button_PLC_Functional_Test_22 := #_w1 AND #In_Functional_Test.Button_PLC_Functional_Test_22;
   #Out_Functional_Test.Electrical_Current_Test_Approved_PLC_Functional_Test_22 := #_w1 AND #In_Functional_Test.Electrical_Current_Test_Approved_PLC_Functional_Test_22;
   #Out_Functional_Test.Visual_Test_Approved_PLC_Functional_Test_22 := #_w1 AND #In_Functional_Test.Visual_Test_Approved_PLC_Functional_Test_22;
   IF #_w1 THEN
       #Out_Functional_Test.Electrical_Current_Read_PLC_Functional_Test_22 := #In_Functional_Test.Electrical_Current_Read_PLC_Functional_Test_22;
   END_IF;
   #Out_Functional_Test.Life_Trigger_PLC_Functional_Test_24 := #_w1 AND #In_Functional_Test.Life_Trigger_PLC_Functional_Test_24;
   #Out_Functional_Test.Star_Test_PLC_Functional_Test_24 := #_w1 AND #In_Functional_Test.Star_Test_PLC_Functional_Test_24;
   #Out_Functional_Test.Button_PLC_Functional_Test_24 := #_w1 AND #In_Functional_Test.Button_PLC_Functional_Test_24;
   #Out_Functional_Test.Electrical_Current_Test_Approved_PLC_Functional_Test_24 := #_w1 AND #In_Functional_Test.Electrical_Current_Test_Approved_PLC_Functional_Test_24;
   #Out_Functional_Test.Visual_Test_Approved_PLC_Functional_Test_24 := #_w1 AND #In_Functional_Test.Visual_Test_Approved_PLC_Functional_Test_24;
   IF #_w1 THEN
       #Out_Functional_Test.Electrical_Current_Read_PLC_Functional_Test_24 := #In_Functional_Test.Electrical_Current_Read_PLC_Functional_Test_24;
   END_IF;
   #Out_Functional_Test.Life_Trigger_PLC_Functional_Test_26 := #_w1 AND #In_Functional_Test.Life_Trigger_PLC_Functional_Test_26;
   #Out_Functional_Test.Star_Test_PLC_Functional_Test_26 := #_w1 AND #In_Functional_Test.Star_Test_PLC_Functional_Test_26;
   #Out_Functional_Test.Button_PLC_Functional_Test_26 := #_w1 AND #In_Functional_Test.Button_PLC_Functional_Test_26;
   #Out_Functional_Test.Electrical_Current_Test_Approved_PLC_Functional_Test_26 := #_w1 AND #In_Functional_Test.Electrical_Current_Test_Approved_PLC_Functional_Test_26;
   #Out_Functional_Test.Visual_Test_Approved_PLC_Functional_Test_26 := #_w1 AND #In_Functional_Test.Visual_Test_Approved_PLC_Functional_Test_26;
   IF #_w1 THEN
       #Out_Functional_Test.Electrical_Current_Read_PLC_Functional_Test_26 := #In_Functional_Test.Electrical_Current_Read_PLC_Functional_Test_26;
   END_IF;
   #Out_Functional_Test.Life_Trigger_PLC_Functional_Test_28 := #_w1 AND #In_Functional_Test.Life_Trigger_PLC_Functional_Test_28;
   #Out_Functional_Test.Star_Test_PLC_Functional_Test_28 := #_w1 AND #In_Functional_Test.Star_Test_PLC_Functional_Test_28;
   #Out_Functional_Test.Button_PLC_Functional_Test_28 := #_w1 AND #In_Functional_Test.Button_PLC_Functional_Test_28;
   #Out_Functional_Test.Electrical_Current_Test_Approved_PLC_Functional_Test_28 := #_w1 AND #In_Functional_Test.Electrical_Current_Test_Approved_PLC_Functional_Test_28;
   #Out_Functional_Test.Visual_Test_Approved_PLC_Functional_Test_28 := #_w1 AND #In_Functional_Test.Visual_Test_Approved_PLC_Functional_Test_28;
   IF #_w1 THEN
       #Out_Functional_Test.Electrical_Current_Read_PLC_Functional_Test_28 := #In_Functional_Test.Electrical_Current_Read_PLC_Functional_Test_28;
   END_IF;
   #Out_Functional_Test.Life_Trigger_PLC_Functional_Test_30 := #_w1 AND #In_Functional_Test.Life_Trigger_PLC_Functional_Test_30;
   #Out_Functional_Test.Star_Test_PLC_Functional_Test_30 := #_w1 AND #In_Functional_Test.Star_Test_PLC_Functional_Test_30;
   #Out_Functional_Test.Button_PLC_Functional_Test_30 := #_w1 AND #In_Functional_Test.Button_PLC_Functional_Test_30;
   #Out_Functional_Test.Electrical_Current_Test_Approved_PLC_Functional_Test_30 := #_w1 AND #In_Functional_Test.Electrical_Current_Test_Approved_PLC_Functional_Test_30;
   #Out_Functional_Test.Visual_Test_Approved_PLC_Functional_Test_30 := #_w1 AND #In_Functional_Test.Visual_Test_Approved_PLC_Functional_Test_30;
   IF #_w1 THEN
       #Out_Functional_Test.Electrical_Current_Read_PLC_Functional_Test_30 := #In_Functional_Test.Electrical_Current_Read_PLC_Functional_Test_30;
   END_IF;
END_REGION

REGION Network 3: Functional Test Station 4
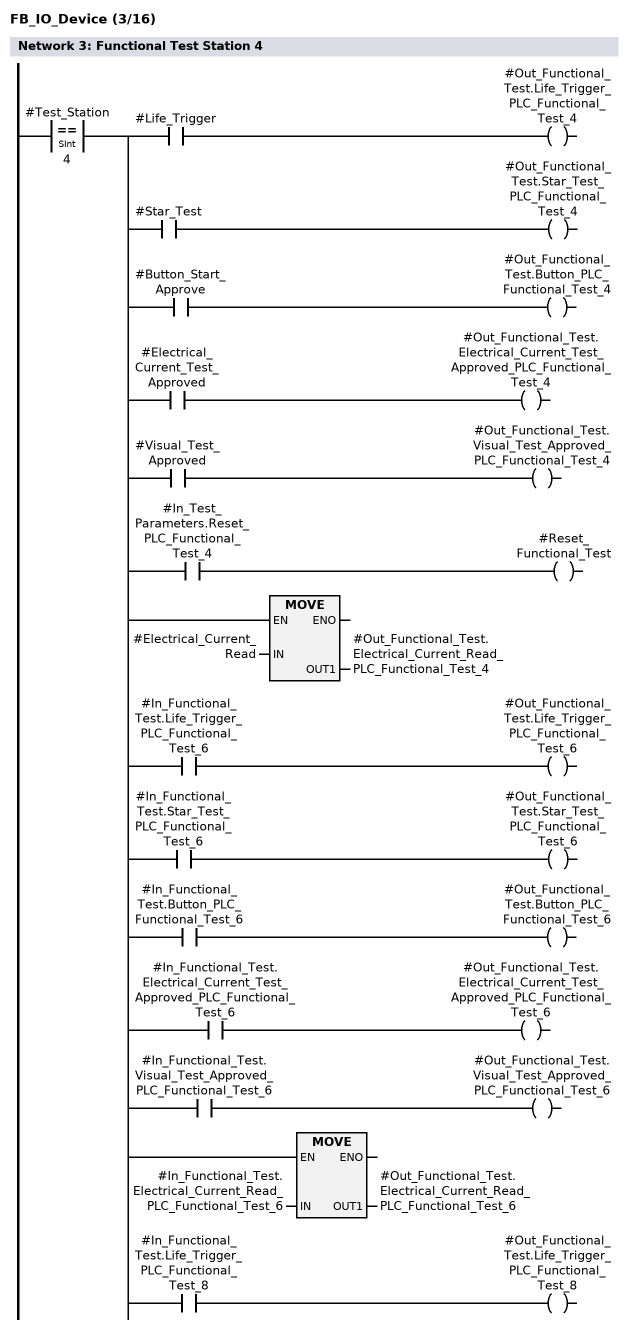
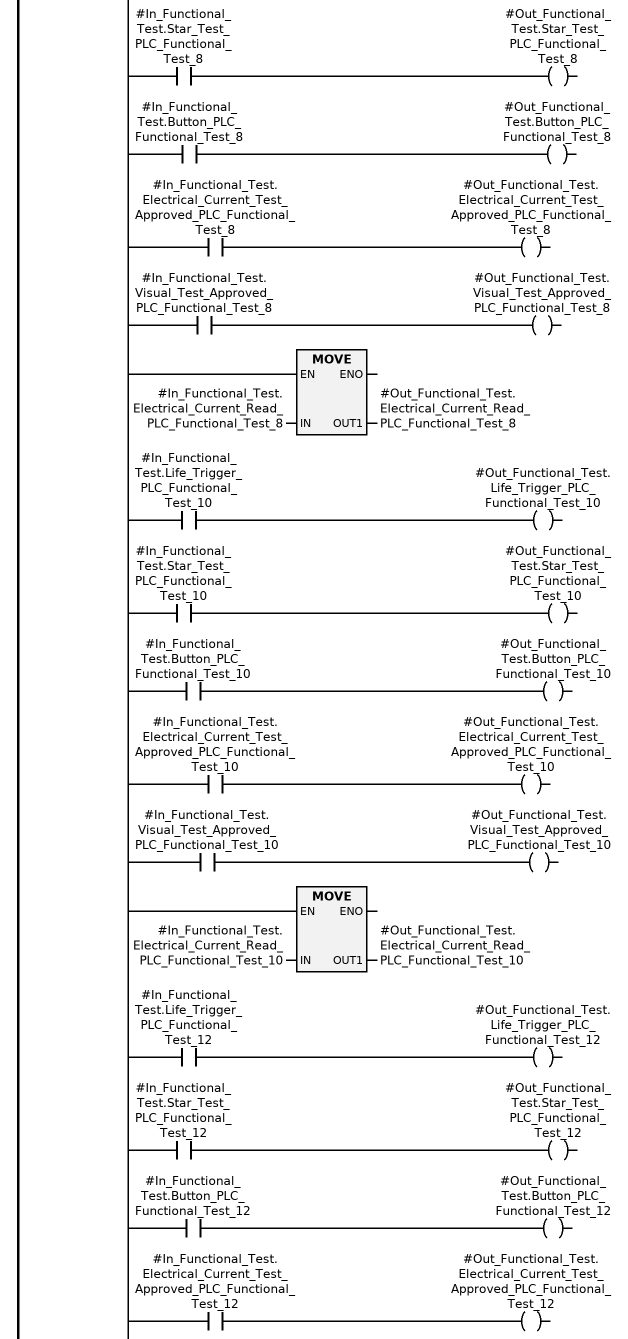
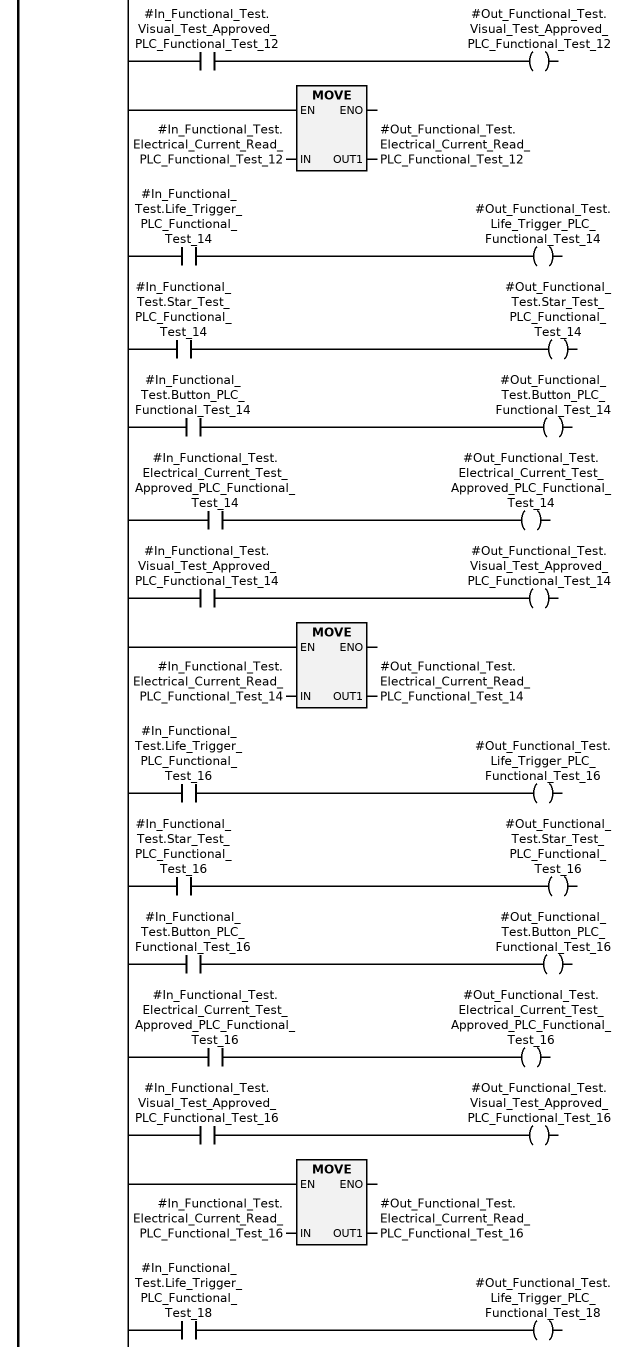
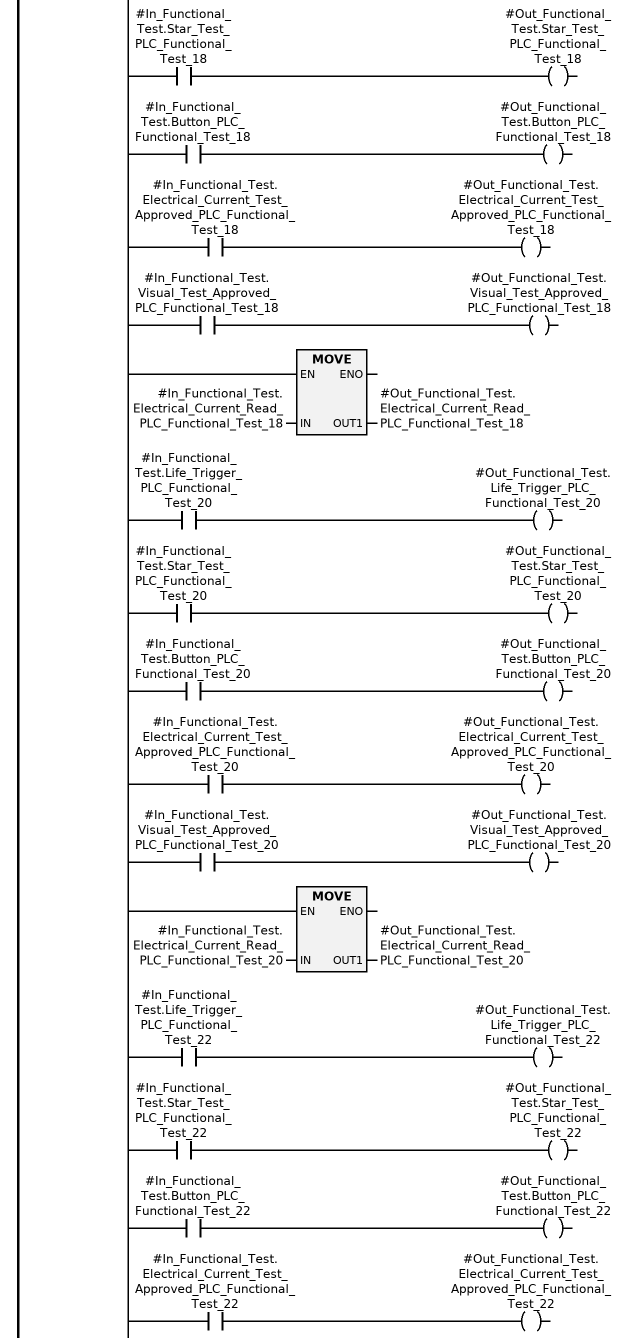
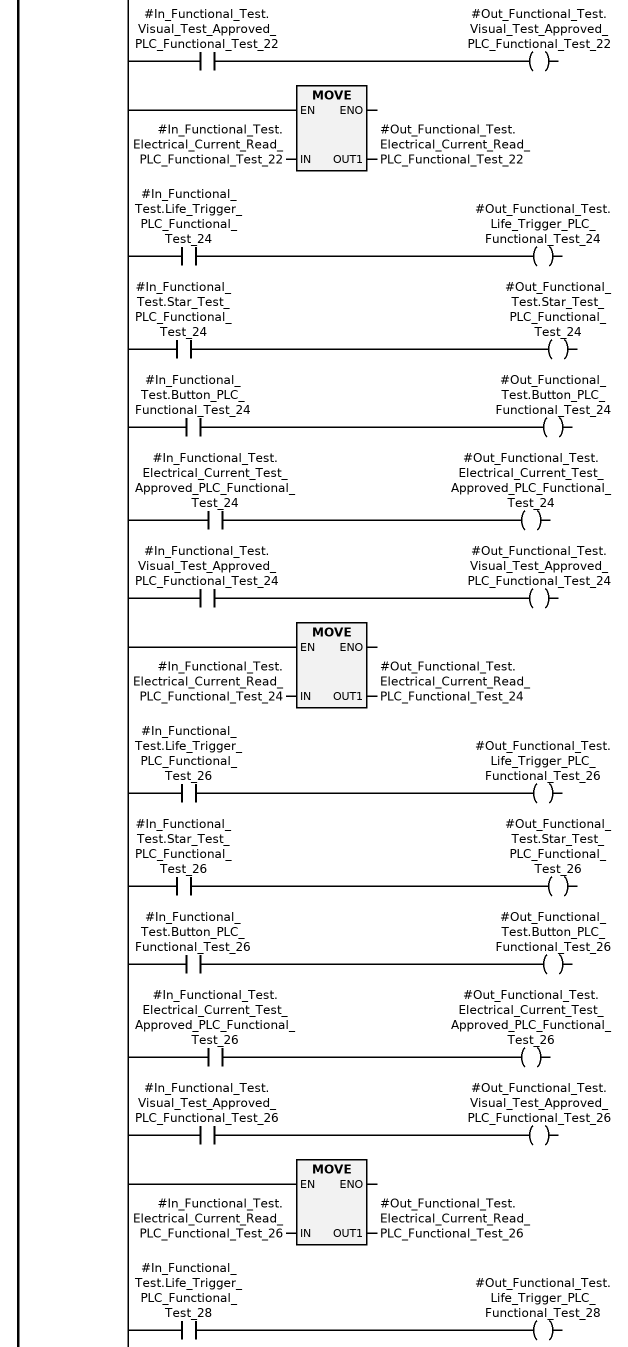
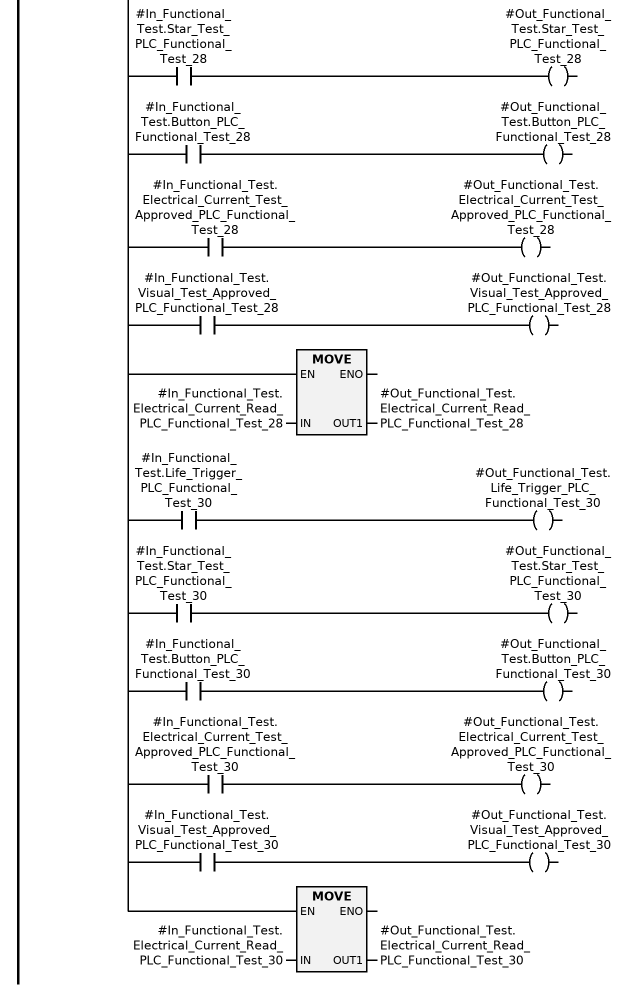
   RUNG wire#powerrail
      { S7_Templates := "SrcType := SInt" } EQ_Contact(in1 := #Test_Station, in2 := 4)
      wire#w1
      Contact( #Life_Trigger )
      Coil( #Out_Functional_Test.Life_Trigger_PLC_Functional_Test_4 )
   END_RUNG
   RUNG wire#w1
      Contact( #Star_Test )
      Coil( #Out_Functional_Test.Star_Test_PLC_Functional_Test_4 )
   END_RUNG
   RUNG wire#w1
      Contact( #Button_Start_Approve )
      Coil( #Out_Functional_Test.Button_PLC_Functional_Test_4 )
   END_RUNG
   RUNG wire#w1
      Contact( #Electrical_Current_Test_Approved )
      Coil( #Out_Functional_Test.Electrical_Current_Test_Approved_PLC_Functional_Test_4 )
   END_RUNG
   RUNG wire#w1
      Contact( #Visual_Test_Approved )
      Coil( #Out_Functional_Test.Visual_Test_Approved_PLC_Functional_Test_4 )
   END_RUNG
   RUNG wire#w1
      Contact( #In_Test_Parameters.Reset_PLC_Functional_Test_4 )
      Coil( #Reset_Functional_Test )
   END_RUNG
   RUNG wire#w1
      Move(in := #Electrical_Current_Read, out1 => #Out_Functional_Test.Electrical_Current_Read_PLC_Functional_Test_4)
   END_RUNG
   RUNG wire#w1
      Contact( #In_Functional_Test.Life_Trigger_PLC_Functional_Test_6 )
      Coil( #Out_Functional_Test.Life_Trigger_PLC_Functional_Test_6 )
   END_RUNG
   RUNG wire#w1
      Contact( #In_Functional_Test.Star_Test_PLC_Functional_Test_6 )
      Coil( #Out_Functional_Test.Star_Test_PLC_Functional_Test_6 )
   END_RUNG
   RUNG wire#w1
      Contact( #In_Functional_Test.Button_PLC_Functional_Test_6 )
      Coil( #Out_Functional_Test.Button_PLC_Functional_Test_6 )
   END_RUNG
   RUNG wire#w1
      Contact( #In_Functional_Test.Electrical_Current_Test_Approved_PLC_Functional_Test_6 )
      Coil( #Out_Functional_Test.Electrical_Current_Test_Approved_PLC_Functional_Test_6 )
   END_RUNG
   RUNG wire#w1
      Contact( #In_Functional_Test.Visual_Test_Approved_PLC_Functional_Test_6 )
      Coil( #Out_Functional_Test.Visual_Test_Approved_PLC_Functional_Test_6 )
   END_RUNG
   RUNG wire#w1
      Move(in := #In_Functional_Test.Electrical_Current_Read_PLC_Functional_Test_6, out1 => #Out_Functional_Test.Electrical_Current_Read_PLC_Functional_Test_6)
   END_RUNG
   RUNG wire#w1
      Contact( #In_Functional_Test.Life_Trigger_PLC_Functional_Test_8 )
      Coil( #Out_Functional_Test.Life_Trigger_PLC_Functional_Test_8 )
   END_RUNG
   RUNG wire#w1
      Contact( #In_Functional_Test.Star_Test_PLC_Functional_Test_8 )
      Coil( #Out_Functional_Test.Star_Test_PLC_Functional_Test_8 )
   END_RUNG
   RUNG wire#w1
      Contact( #In_Functional_Test.Button_PLC_Functional_Test_8 )
      Coil( #Out_Functional_Test.Button_PLC_Functional_Test_8 )
   END_RUNG
   RUNG wire#w1
      Contact( #In_Functional_Test.Electrical_Current_Test_Approved_PLC_Functional_Test_8 )
      Coil( #Out_Functional_Test.Electrical_Current_Test_Approved_PLC_Functional_Test_8 )
   END_RUNG
   RUNG wire#w1
      Contact( #In_Functional_Test.Visual_Test_Approved_PLC_Functional_Test_8 )
      Coil( #Out_Functional_Test.Visual_Test_Approved_PLC_Functional_Test_8 )
   END_RUNG
   RUNG wire#w1
      Move(in := #In_Functional_Test.Electrical_Current_Read_PLC_Functional_Test_8, out1 => #Out_Functional_Test.Electrical_Current_Read_PLC_Functional_Test_8)
   END_RUNG
   RUNG wire#w1
      Contact( #In_Functional_Test.Life_Trigger_PLC_Functional_Test_10 )
      Coil( #Out_Functional_Test.Life_Trigger_PLC_Functional_Test_10 )
   END_RUNG
   RUNG wire#w1
      Contact( #In_Functional_Test.Star_Test_PLC_Functional_Test_10 )
      Coil( #Out_Functional_Test.Star_Test_PLC_Functional_Test_10 )
   END_RUNG
   RUNG wire#w1
      Contact( #In_Functional_Test.Button_PLC_Functional_Test_10 )
      Coil( #Out_Functional_Test.Button_PLC_Functional_Test_10 )
   END_RUNG
   RUNG wire#w1
      Contact( #In_Functional_Test.Electrical_Current_Test_Approved_PLC_Functional_Test_10 )
      Coil( #Out_Functional_Test.Electrical_Current_Test_Approved_PLC_Functional_Test_10 )
   END_RUNG
   RUNG wire#w1
      Contact( #In_Functional_Test.Visual_Test_Approved_PLC_Functional_Test_10 )
      Coil( #Out_Functional_Test.Visual_Test_Approved_PLC_Functional_Test_10 )
   END_RUNG
   RUNG wire#w1
      Move(in := #In_Functional_Test.Electrical_Current_Read_PLC_Functional_Test_10, out1 => #Out_Functional_Test.Electrical_Current_Read_PLC_Functional_Test_10)
   END_RUNG
   RUNG wire#w1
      Contact( #In_Functional_Test.Life_Trigger_PLC_Functional_Test_12 )
      Coil( #Out_Functional_Test.Life_Trigger_PLC_Functional_Test_12 )
   END_RUNG
   RUNG wire#w1
      Contact( #In_Functional_Test.Star_Test_PLC_Functional_Test_12 )
      Coil( #Out_Functional_Test.Star_Test_PLC_Functional_Test_12 )
   END_RUNG
   RUNG wire#w1
      Contact( #In_Functional_Test.Button_PLC_Functional_Test_12 )
      Coil( #Out_Functional_Test.Button_PLC_Functional_Test_12 )
   END_RUNG
   RUNG wire#w1
      Contact( #In_Functional_Test.Electrical_Current_Test_Approved_PLC_Functional_Test_12 )
      Coil( #Out_Functional_Test.Electrical_Current_Test_Approved_PLC_Functional_Test_12 )
   END_RUNG
   RUNG wire#w1
      Contact( #In_Functional_Test.Visual_Test_Approved_PLC_Functional_Test_12 )
      Coil( #Out_Functional_Test.Visual_Test_Approved_PLC_Functional_Test_12 )
   END_RUNG
   RUNG wire#w1
      Move(in := #In_Functional_Test.Electrical_Current_Read_PLC_Functional_Test_12, out1 => #Out_Functional_Test.Electrical_Current_Read_PLC_Functional_Test_12)
   END_RUNG
   RUNG wire#w1
      Contact( #In_Functional_Test.Life_Trigger_PLC_Functional_Test_14 )
      Coil( #Out_Functional_Test.Life_Trigger_PLC_Functional_Test_14 )
   END_RUNG
   RUNG wire#w1
      Contact( #In_Functional_Test.Star_Test_PLC_Functional_Test_14 )
      Coil( #Out_Functional_Test.Star_Test_PLC_Functional_Test_14 )
   END_RUNG
   RUNG wire#w1
      Contact( #In_Functional_Test.Button_PLC_Functional_Test_14 )
      Coil( #Out_Functional_Test.Button_PLC_Functional_Test_14 )
   END_RUNG
   RUNG wire#w1
      Contact( #In_Functional_Test.Electrical_Current_Test_Approved_PLC_Functional_Test_14 )
      Coil( #Out_Functional_Test.Electrical_Current_Test_Approved_PLC_Functional_Test_14 )
   END_RUNG
   RUNG wire#w1
      Contact( #In_Functional_Test.Visual_Test_Approved_PLC_Functional_Test_14 )
      Coil( #Out_Functional_Test.Visual_Test_Approved_PLC_Functional_Test_14 )
   END_RUNG
   RUNG wire#w1
      Move(in := #In_Functional_Test.Electrical_Current_Read_PLC_Functional_Test_14, out1 => #Out_Functional_Test.Electrical_Current_Read_PLC_Functional_Test_14)
   END_RUNG
   RUNG wire#w1
      Contact( #In_Functional_Test.Life_Trigger_PLC_Functional_Test_16 )
      Coil( #Out_Functional_Test.Life_Trigger_PLC_Functional_Test_16 )
   END_RUNG
   RUNG wire#w1
      Contact( #In_Functional_Test.Star_Test_PLC_Functional_Test_16 )
      Coil( #Out_Functional_Test.Star_Test_PLC_Functional_Test_16 )
   END_RUNG
   RUNG wire#w1
      Contact( #In_Functional_Test.Button_PLC_Functional_Test_16 )
      Coil( #Out_Functional_Test.Button_PLC_Functional_Test_16 )
   END_RUNG
   RUNG wire#w1
      Contact( #In_Functional_Test.Electrical_Current_Test_Approved_PLC_Functional_Test_16 )
      Coil( #Out_Functional_Test.Electrical_Current_Test_Approved_PLC_Functional_Test_16 )
   END_RUNG
   RUNG wire#w1
      Contact( #In_Functional_Test.Visual_Test_Approved_PLC_Functional_Test_16 )
      Coil( #Out_Functional_Test.Visual_Test_Approved_PLC_Functional_Test_16 )
   END_RUNG
   RUNG wire#w1
      Move(in := #In_Functional_Test.Electrical_Current_Read_PLC_Functional_Test_16, out1 => #Out_Functional_Test.Electrical_Current_Read_PLC_Functional_Test_16)
   END_RUNG
   RUNG wire#w1
      Contact( #In_Functional_Test.Life_Trigger_PLC_Functional_Test_18 )
      Coil( #Out_Functional_Test.Life_Trigger_PLC_Functional_Test_18 )
   END_RUNG
   RUNG wire#w1
      Contact( #In_Functional_Test.Star_Test_PLC_Functional_Test_18 )
      Coil( #Out_Functional_Test.Star_Test_PLC_Functional_Test_18 )
   END_RUNG
   RUNG wire#w1
      Contact( #In_Functional_Test.Button_PLC_Functional_Test_18 )
      Coil( #Out_Functional_Test.Button_PLC_Functional_Test_18 )
   END_RUNG
   RUNG wire#w1
      Contact( #In_Functional_Test.Electrical_Current_Test_Approved_PLC_Functional_Test_18 )
      Coil( #Out_Functional_Test.Electrical_Current_Test_Approved_PLC_Functional_Test_18 )
   END_RUNG
   RUNG wire#w1
      Contact( #In_Functional_Test.Visual_Test_Approved_PLC_Functional_Test_18 )
      Coil( #Out_Functional_Test.Visual_Test_Approved_PLC_Functional_Test_18 )
   END_RUNG
   RUNG wire#w1
      Move(in := #In_Functional_Test.Electrical_Current_Read_PLC_Functional_Test_18, out1 => #Out_Functional_Test.Electrical_Current_Read_PLC_Functional_Test_18)
   END_RUNG
   RUNG wire#w1
      Contact( #In_Functional_Test.Life_Trigger_PLC_Functional_Test_20 )
      Coil( #Out_Functional_Test.Life_Trigger_PLC_Functional_Test_20 )
   END_RUNG
   RUNG wire#w1
      Contact( #In_Functional_Test.Star_Test_PLC_Functional_Test_20 )
      Coil( #Out_Functional_Test.Star_Test_PLC_Functional_Test_20 )
   END_RUNG
   RUNG wire#w1
      Contact( #In_Functional_Test.Button_PLC_Functional_Test_20 )
      Coil( #Out_Functional_Test.Button_PLC_Functional_Test_20 )
   END_RUNG
   RUNG wire#w1
      Contact( #In_Functional_Test.Electrical_Current_Test_Approved_PLC_Functional_Test_20 )
      Coil( #Out_Functional_Test.Electrical_Current_Test_Approved_PLC_Functional_Test_20 )
   END_RUNG
   RUNG wire#w1
      Contact( #In_Functional_Test.Visual_Test_Approved_PLC_Functional_Test_20 )
      Coil( #Out_Functional_Test.Visual_Test_Approved_PLC_Functional_Test_20 )
   END_RUNG
   RUNG wire#w1
      Move(in := #In_Functional_Test.Electrical_Current_Read_PLC_Functional_Test_20, out1 => #Out_Functional_Test.Electrical_Current_Read_PLC_Functional_Test_20)
   END_RUNG
   RUNG wire#w1
      Contact( #In_Functional_Test.Life_Trigger_PLC_Functional_Test_22 )
      Coil( #Out_Functional_Test.Life_Trigger_PLC_Functional_Test_22 )
   END_RUNG
   RUNG wire#w1
      Contact( #In_Functional_Test.Star_Test_PLC_Functional_Test_22 )
      Coil( #Out_Functional_Test.Star_Test_PLC_Functional_Test_22 )
   END_RUNG
   RUNG wire#w1
      Contact( #In_Functional_Test.Button_PLC_Functional_Test_22 )
      Coil( #Out_Functional_Test.Button_PLC_Functional_Test_22 )
   END_RUNG
   RUNG wire#w1
      Contact( #In_Functional_Test.Electrical_Current_Test_Approved_PLC_Functional_Test_22 )
      Coil( #Out_Functional_Test.Electrical_Current_Test_Approved_PLC_Functional_Test_22 )
   END_RUNG
   RUNG wire#w1
      Contact( #In_Functional_Test.Visual_Test_Approved_PLC_Functional_Test_22 )
      Coil( #Out_Functional_Test.Visual_Test_Approved_PLC_Functional_Test_22 )
   END_RUNG
   RUNG wire#w1
      Move(in := #In_Functional_Test.Electrical_Current_Read_PLC_Functional_Test_22, out1 => #Out_Functional_Test.Electrical_Current_Read_PLC_Functional_Test_22)
   END_RUNG
   RUNG wire#w1
      Contact( #In_Functional_Test.Life_Trigger_PLC_Functional_Test_24 )
      Coil( #Out_Functional_Test.Life_Trigger_PLC_Functional_Test_24 )
   END_RUNG
   RUNG wire#w1
      Contact( #In_Functional_Test.Star_Test_PLC_Functional_Test_24 )
      Coil( #Out_Functional_Test.Star_Test_PLC_Functional_Test_24 )
   END_RUNG
   RUNG wire#w1
      Contact( #In_Functional_Test.Button_PLC_Functional_Test_24 )
      Coil( #Out_Functional_Test.Button_PLC_Functional_Test_24 )
   END_RUNG
   RUNG wire#w1
      Contact( #In_Functional_Test.Electrical_Current_Test_Approved_PLC_Functional_Test_24 )
      Coil( #Out_Functional_Test.Electrical_Current_Test_Approved_PLC_Functional_Test_24 )
   END_RUNG
   RUNG wire#w1
      Contact( #In_Functional_Test.Visual_Test_Approved_PLC_Functional_Test_24 )
      Coil( #Out_Functional_Test.Visual_Test_Approved_PLC_Functional_Test_24 )
   END_RUNG
   RUNG wire#w1
      Move(in := #In_Functional_Test.Electrical_Current_Read_PLC_Functional_Test_24, out1 => #Out_Functional_Test.Electrical_Current_Read_PLC_Functional_Test_24)
   END_RUNG
   RUNG wire#w1
      Contact( #In_Functional_Test.Life_Trigger_PLC_Functional_Test_26 )
      Coil( #Out_Functional_Test.Life_Trigger_PLC_Functional_Test_26 )
   END_RUNG
   RUNG wire#w1
      Contact( #In_Functional_Test.Star_Test_PLC_Functional_Test_26 )
      Coil( #Out_Functional_Test.Star_Test_PLC_Functional_Test_26 )
   END_RUNG
   RUNG wire#w1
      Contact( #In_Functional_Test.Button_PLC_Functional_Test_26 )
      Coil( #Out_Functional_Test.Button_PLC_Functional_Test_26 )
   END_RUNG
   RUNG wire#w1
      Contact( #In_Functional_Test.Electrical_Current_Test_Approved_PLC_Functional_Test_26 )
      Coil( #Out_Functional_Test.Electrical_Current_Test_Approved_PLC_Functional_Test_26 )
   END_RUNG
   RUNG wire#w1
      Contact( #In_Functional_Test.Visual_Test_Approved_PLC_Functional_Test_26 )
      Coil( #Out_Functional_Test.Visual_Test_Approved_PLC_Functional_Test_26 )
   END_RUNG
   RUNG wire#w1
      Move(in := #In_Functional_Test.Electrical_Current_Read_PLC_Functional_Test_26, out1 => #Out_Functional_Test.Electrical_Current_Read_PLC_Functional_Test_26)
   END_RUNG
   RUNG wire#w1
      Contact( #In_Functional_Test.Life_Trigger_PLC_Functional_Test_28 )
      Coil( #Out_Functional_Test.Life_Trigger_PLC_Functional_Test_28 )
   END_RUNG
   RUNG wire#w1
      Contact( #In_Functional_Test.Star_Test_PLC_Functional_Test_28 )
      Coil( #Out_Functional_Test.Star_Test_PLC_Functional_Test_28 )
   END_RUNG
   RUNG wire#w1
      Contact( #In_Functional_Test.Button_PLC_Functional_Test_28 )
      Coil( #Out_Functional_Test.Button_PLC_Functional_Test_28 )
   END_RUNG
   RUNG wire#w1
      Contact( #In_Functional_Test.Electrical_Current_Test_Approved_PLC_Functional_Test_28 )
      Coil( #Out_Functional_Test.Electrical_Current_Test_Approved_PLC_Functional_Test_28 )
   END_RUNG
   RUNG wire#w1
      Contact( #In_Functional_Test.Visual_Test_Approved_PLC_Functional_Test_28 )
      Coil( #Out_Functional_Test.Visual_Test_Approved_PLC_Functional_Test_28 )
   END_RUNG
   RUNG wire#w1
      Move(in := #In_Functional_Test.Electrical_Current_Read_PLC_Functional_Test_28, out1 => #Out_Functional_Test.Electrical_Current_Read_PLC_Functional_Test_28)
   END_RUNG
   RUNG wire#w1
      Contact( #In_Functional_Test.Life_Trigger_PLC_Functional_Test_30 )
      Coil( #Out_Functional_Test.Life_Trigger_PLC_Functional_Test_30 )
   END_RUNG
   RUNG wire#w1
      Contact( #In_Functional_Test.Star_Test_PLC_Functional_Test_30 )
      Coil( #Out_Functional_Test.Star_Test_PLC_Functional_Test_30 )
   END_RUNG
   RUNG wire#w1
      Contact( #In_Functional_Test.Button_PLC_Functional_Test_30 )
      Coil( #Out_Functional_Test.Button_PLC_Functional_Test_30 )
   END_RUNG
   RUNG wire#w1
      Contact( #In_Functional_Test.Electrical_Current_Test_Approved_PLC_Functional_Test_30 )
      Coil( #Out_Functional_Test.Electrical_Current_Test_Approved_PLC_Functional_Test_30 )
   END_RUNG
   RUNG wire#w1
      Contact( #In_Functional_Test.Visual_Test_Approved_PLC_Functional_Test_30 )
      Coil( #Out_Functional_Test.Visual_Test_Approved_PLC_Functional_Test_30 )
   END_RUNG
   RUNG wire#w1
      Move(in := #In_Functional_Test.Electrical_Current_Read_PLC_Functional_Test_30, out1 => #Out_Functional_Test.Electrical_Current_Read_PLC_Functional_Test_30)
   END_RUNG
   // the same network as SCL:
   #_w1 := #Test_Station = 4;
   #Out_Functional_Test.Life_Trigger_PLC_Functional_Test_4 := #_w1 AND #Life_Trigger;
   #Out_Functional_Test.Star_Test_PLC_Functional_Test_4 := #_w1 AND #Star_Test;
   #Out_Functional_Test.Button_PLC_Functional_Test_4 := #_w1 AND #Button_Start_Approve;
   #Out_Functional_Test.Electrical_Current_Test_Approved_PLC_Functional_Test_4 := #_w1 AND #Electrical_Current_Test_Approved;
   #Out_Functional_Test.Visual_Test_Approved_PLC_Functional_Test_4 := #_w1 AND #Visual_Test_Approved;
   #Reset_Functional_Test := #_w1 AND #In_Test_Parameters.Reset_PLC_Functional_Test_4;
   IF #_w1 THEN
       #Out_Functional_Test.Electrical_Current_Read_PLC_Functional_Test_4 := #Electrical_Current_Read;
   END_IF;
   #Out_Functional_Test.Life_Trigger_PLC_Functional_Test_6 := #_w1 AND #In_Functional_Test.Life_Trigger_PLC_Functional_Test_6;
   #Out_Functional_Test.Star_Test_PLC_Functional_Test_6 := #_w1 AND #In_Functional_Test.Star_Test_PLC_Functional_Test_6;
   #Out_Functional_Test.Button_PLC_Functional_Test_6 := #_w1 AND #In_Functional_Test.Button_PLC_Functional_Test_6;
   #Out_Functional_Test.Electrical_Current_Test_Approved_PLC_Functional_Test_6 := #_w1 AND #In_Functional_Test.Electrical_Current_Test_Approved_PLC_Functional_Test_6;
   #Out_Functional_Test.Visual_Test_Approved_PLC_Functional_Test_6 := #_w1 AND #In_Functional_Test.Visual_Test_Approved_PLC_Functional_Test_6;
   IF #_w1 THEN
       #Out_Functional_Test.Electrical_Current_Read_PLC_Functional_Test_6 := #In_Functional_Test.Electrical_Current_Read_PLC_Functional_Test_6;
   END_IF;
   #Out_Functional_Test.Life_Trigger_PLC_Functional_Test_8 := #_w1 AND #In_Functional_Test.Life_Trigger_PLC_Functional_Test_8;
   #Out_Functional_Test.Star_Test_PLC_Functional_Test_8 := #_w1 AND #In_Functional_Test.Star_Test_PLC_Functional_Test_8;
   #Out_Functional_Test.Button_PLC_Functional_Test_8 := #_w1 AND #In_Functional_Test.Button_PLC_Functional_Test_8;
   #Out_Functional_Test.Electrical_Current_Test_Approved_PLC_Functional_Test_8 := #_w1 AND #In_Functional_Test.Electrical_Current_Test_Approved_PLC_Functional_Test_8;
   #Out_Functional_Test.Visual_Test_Approved_PLC_Functional_Test_8 := #_w1 AND #In_Functional_Test.Visual_Test_Approved_PLC_Functional_Test_8;
   IF #_w1 THEN
       #Out_Functional_Test.Electrical_Current_Read_PLC_Functional_Test_8 := #In_Functional_Test.Electrical_Current_Read_PLC_Functional_Test_8;
   END_IF;
   #Out_Functional_Test.Life_Trigger_PLC_Functional_Test_10 := #_w1 AND #In_Functional_Test.Life_Trigger_PLC_Functional_Test_10;
   #Out_Functional_Test.Star_Test_PLC_Functional_Test_10 := #_w1 AND #In_Functional_Test.Star_Test_PLC_Functional_Test_10;
   #Out_Functional_Test.Button_PLC_Functional_Test_10 := #_w1 AND #In_Functional_Test.Button_PLC_Functional_Test_10;
   #Out_Functional_Test.Electrical_Current_Test_Approved_PLC_Functional_Test_10 := #_w1 AND #In_Functional_Test.Electrical_Current_Test_Approved_PLC_Functional_Test_10;
   #Out_Functional_Test.Visual_Test_Approved_PLC_Functional_Test_10 := #_w1 AND #In_Functional_Test.Visual_Test_Approved_PLC_Functional_Test_10;
   IF #_w1 THEN
       #Out_Functional_Test.Electrical_Current_Read_PLC_Functional_Test_10 := #In_Functional_Test.Electrical_Current_Read_PLC_Functional_Test_10;
   END_IF;
   #Out_Functional_Test.Life_Trigger_PLC_Functional_Test_12 := #_w1 AND #In_Functional_Test.Life_Trigger_PLC_Functional_Test_12;
   #Out_Functional_Test.Star_Test_PLC_Functional_Test_12 := #_w1 AND #In_Functional_Test.Star_Test_PLC_Functional_Test_12;
   #Out_Functional_Test.Button_PLC_Functional_Test_12 := #_w1 AND #In_Functional_Test.Button_PLC_Functional_Test_12;
   #Out_Functional_Test.Electrical_Current_Test_Approved_PLC_Functional_Test_12 := #_w1 AND #In_Functional_Test.Electrical_Current_Test_Approved_PLC_Functional_Test_12;
   #Out_Functional_Test.Visual_Test_Approved_PLC_Functional_Test_12 := #_w1 AND #In_Functional_Test.Visual_Test_Approved_PLC_Functional_Test_12;
   IF #_w1 THEN
       #Out_Functional_Test.Electrical_Current_Read_PLC_Functional_Test_12 := #In_Functional_Test.Electrical_Current_Read_PLC_Functional_Test_12;
   END_IF;
   #Out_Functional_Test.Life_Trigger_PLC_Functional_Test_14 := #_w1 AND #In_Functional_Test.Life_Trigger_PLC_Functional_Test_14;
   #Out_Functional_Test.Star_Test_PLC_Functional_Test_14 := #_w1 AND #In_Functional_Test.Star_Test_PLC_Functional_Test_14;
   #Out_Functional_Test.Button_PLC_Functional_Test_14 := #_w1 AND #In_Functional_Test.Button_PLC_Functional_Test_14;
   #Out_Functional_Test.Electrical_Current_Test_Approved_PLC_Functional_Test_14 := #_w1 AND #In_Functional_Test.Electrical_Current_Test_Approved_PLC_Functional_Test_14;
   #Out_Functional_Test.Visual_Test_Approved_PLC_Functional_Test_14 := #_w1 AND #In_Functional_Test.Visual_Test_Approved_PLC_Functional_Test_14;
   IF #_w1 THEN
       #Out_Functional_Test.Electrical_Current_Read_PLC_Functional_Test_14 := #In_Functional_Test.Electrical_Current_Read_PLC_Functional_Test_14;
   END_IF;
   #Out_Functional_Test.Life_Trigger_PLC_Functional_Test_16 := #_w1 AND #In_Functional_Test.Life_Trigger_PLC_Functional_Test_16;
   #Out_Functional_Test.Star_Test_PLC_Functional_Test_16 := #_w1 AND #In_Functional_Test.Star_Test_PLC_Functional_Test_16;
   #Out_Functional_Test.Button_PLC_Functional_Test_16 := #_w1 AND #In_Functional_Test.Button_PLC_Functional_Test_16;
   #Out_Functional_Test.Electrical_Current_Test_Approved_PLC_Functional_Test_16 := #_w1 AND #In_Functional_Test.Electrical_Current_Test_Approved_PLC_Functional_Test_16;
   #Out_Functional_Test.Visual_Test_Approved_PLC_Functional_Test_16 := #_w1 AND #In_Functional_Test.Visual_Test_Approved_PLC_Functional_Test_16;
   IF #_w1 THEN
       #Out_Functional_Test.Electrical_Current_Read_PLC_Functional_Test_16 := #In_Functional_Test.Electrical_Current_Read_PLC_Functional_Test_16;
   END_IF;
   #Out_Functional_Test.Life_Trigger_PLC_Functional_Test_18 := #_w1 AND #In_Functional_Test.Life_Trigger_PLC_Functional_Test_18;
   #Out_Functional_Test.Star_Test_PLC_Functional_Test_18 := #_w1 AND #In_Functional_Test.Star_Test_PLC_Functional_Test_18;
   #Out_Functional_Test.Button_PLC_Functional_Test_18 := #_w1 AND #In_Functional_Test.Button_PLC_Functional_Test_18;
   #Out_Functional_Test.Electrical_Current_Test_Approved_PLC_Functional_Test_18 := #_w1 AND #In_Functional_Test.Electrical_Current_Test_Approved_PLC_Functional_Test_18;
   #Out_Functional_Test.Visual_Test_Approved_PLC_Functional_Test_18 := #_w1 AND #In_Functional_Test.Visual_Test_Approved_PLC_Functional_Test_18;
   IF #_w1 THEN
       #Out_Functional_Test.Electrical_Current_Read_PLC_Functional_Test_18 := #In_Functional_Test.Electrical_Current_Read_PLC_Functional_Test_18;
   END_IF;
   #Out_Functional_Test.Life_Trigger_PLC_Functional_Test_20 := #_w1 AND #In_Functional_Test.Life_Trigger_PLC_Functional_Test_20;
   #Out_Functional_Test.Star_Test_PLC_Functional_Test_20 := #_w1 AND #In_Functional_Test.Star_Test_PLC_Functional_Test_20;
   #Out_Functional_Test.Button_PLC_Functional_Test_20 := #_w1 AND #In_Functional_Test.Button_PLC_Functional_Test_20;
   #Out_Functional_Test.Electrical_Current_Test_Approved_PLC_Functional_Test_20 := #_w1 AND #In_Functional_Test.Electrical_Current_Test_Approved_PLC_Functional_Test_20;
   #Out_Functional_Test.Visual_Test_Approved_PLC_Functional_Test_20 := #_w1 AND #In_Functional_Test.Visual_Test_Approved_PLC_Functional_Test_20;
   IF #_w1 THEN
       #Out_Functional_Test.Electrical_Current_Read_PLC_Functional_Test_20 := #In_Functional_Test.Electrical_Current_Read_PLC_Functional_Test_20;
   END_IF;
   #Out_Functional_Test.Life_Trigger_PLC_Functional_Test_22 := #_w1 AND #In_Functional_Test.Life_Trigger_PLC_Functional_Test_22;
   #Out_Functional_Test.Star_Test_PLC_Functional_Test_22 := #_w1 AND #In_Functional_Test.Star_Test_PLC_Functional_Test_22;
   #Out_Functional_Test.Button_PLC_Functional_Test_22 := #_w1 AND #In_Functional_Test.Button_PLC_Functional_Test_22;
   #Out_Functional_Test.Electrical_Current_Test_Approved_PLC_Functional_Test_22 := #_w1 AND #In_Functional_Test.Electrical_Current_Test_Approved_PLC_Functional_Test_22;
   #Out_Functional_Test.Visual_Test_Approved_PLC_Functional_Test_22 := #_w1 AND #In_Functional_Test.Visual_Test_Approved_PLC_Functional_Test_22;
   IF #_w1 THEN
       #Out_Functional_Test.Electrical_Current_Read_PLC_Functional_Test_22 := #In_Functional_Test.Electrical_Current_Read_PLC_Functional_Test_22;
   END_IF;
   #Out_Functional_Test.Life_Trigger_PLC_Functional_Test_24 := #_w1 AND #In_Functional_Test.Life_Trigger_PLC_Functional_Test_24;
   #Out_Functional_Test.Star_Test_PLC_Functional_Test_24 := #_w1 AND #In_Functional_Test.Star_Test_PLC_Functional_Test_24;
   #Out_Functional_Test.Button_PLC_Functional_Test_24 := #_w1 AND #In_Functional_Test.Button_PLC_Functional_Test_24;
   #Out_Functional_Test.Electrical_Current_Test_Approved_PLC_Functional_Test_24 := #_w1 AND #In_Functional_Test.Electrical_Current_Test_Approved_PLC_Functional_Test_24;
   #Out_Functional_Test.Visual_Test_Approved_PLC_Functional_Test_24 := #_w1 AND #In_Functional_Test.Visual_Test_Approved_PLC_Functional_Test_24;
   IF #_w1 THEN
       #Out_Functional_Test.Electrical_Current_Read_PLC_Functional_Test_24 := #In_Functional_Test.Electrical_Current_Read_PLC_Functional_Test_24;
   END_IF;
   #Out_Functional_Test.Life_Trigger_PLC_Functional_Test_26 := #_w1 AND #In_Functional_Test.Life_Trigger_PLC_Functional_Test_26;
   #Out_Functional_Test.Star_Test_PLC_Functional_Test_26 := #_w1 AND #In_Functional_Test.Star_Test_PLC_Functional_Test_26;
   #Out_Functional_Test.Button_PLC_Functional_Test_26 := #_w1 AND #In_Functional_Test.Button_PLC_Functional_Test_26;
   #Out_Functional_Test.Electrical_Current_Test_Approved_PLC_Functional_Test_26 := #_w1 AND #In_Functional_Test.Electrical_Current_Test_Approved_PLC_Functional_Test_26;
   #Out_Functional_Test.Visual_Test_Approved_PLC_Functional_Test_26 := #_w1 AND #In_Functional_Test.Visual_Test_Approved_PLC_Functional_Test_26;
   IF #_w1 THEN
       #Out_Functional_Test.Electrical_Current_Read_PLC_Functional_Test_26 := #In_Functional_Test.Electrical_Current_Read_PLC_Functional_Test_26;
   END_IF;
   #Out_Functional_Test.Life_Trigger_PLC_Functional_Test_28 := #_w1 AND #In_Functional_Test.Life_Trigger_PLC_Functional_Test_28;
   #Out_Functional_Test.Star_Test_PLC_Functional_Test_28 := #_w1 AND #In_Functional_Test.Star_Test_PLC_Functional_Test_28;
   #Out_Functional_Test.Button_PLC_Functional_Test_28 := #_w1 AND #In_Functional_Test.Button_PLC_Functional_Test_28;
   #Out_Functional_Test.Electrical_Current_Test_Approved_PLC_Functional_Test_28 := #_w1 AND #In_Functional_Test.Electrical_Current_Test_Approved_PLC_Functional_Test_28;
   #Out_Functional_Test.Visual_Test_Approved_PLC_Functional_Test_28 := #_w1 AND #In_Functional_Test.Visual_Test_Approved_PLC_Functional_Test_28;
   IF #_w1 THEN
       #Out_Functional_Test.Electrical_Current_Read_PLC_Functional_Test_28 := #In_Functional_Test.Electrical_Current_Read_PLC_Functional_Test_28;
   END_IF;
   #Out_Functional_Test.Life_Trigger_PLC_Functional_Test_30 := #_w1 AND #In_Functional_Test.Life_Trigger_PLC_Functional_Test_30;
   #Out_Functional_Test.Star_Test_PLC_Functional_Test_30 := #_w1 AND #In_Functional_Test.Star_Test_PLC_Functional_Test_30;
   #Out_Functional_Test.Button_PLC_Functional_Test_30 := #_w1 AND #In_Functional_Test.Button_PLC_Functional_Test_30;
   #Out_Functional_Test.Electrical_Current_Test_Approved_PLC_Functional_Test_30 := #_w1 AND #In_Functional_Test.Electrical_Current_Test_Approved_PLC_Functional_Test_30;
   #Out_Functional_Test.Visual_Test_Approved_PLC_Functional_Test_30 := #_w1 AND #In_Functional_Test.Visual_Test_Approved_PLC_Functional_Test_30;
   IF #_w1 THEN
       #Out_Functional_Test.Electrical_Current_Read_PLC_Functional_Test_30 := #In_Functional_Test.Electrical_Current_Read_PLC_Functional_Test_30;
   END_IF;
END_REGION

